# B&R Automation Studio project x20ost (part 7)

#### bnrdevts.c
```c
/********************************************************************
 * COPYRIGHT -- Kontora
 ********************************************************************
 * Program: bnrmain
 * File: bnrlsens.c
 * Author: Abramenya
 * Created: January 19, 2009
 *******************************************************************/

#include "bnrdevts.h"
#include "bnrmain.h"
#ifdef _DEFAULT_INCLUDES
 #include <AsDefault.h>
#endif
_GLOBAL BYTE nFSignal;
void CDevTS_Init(This,CPin *pPN,BOOL *pTlValue,BYTE byID,BYTE byIID,BYTE byState,BYTE byPriority,BYTE byCRemPulce,BYTE byCSetPulce,BYTE byAlarmMode)
{
    DECLARE_SINGLE_OPEN(CDevTS)
	//memcpy(pTU,&pT->pP,sizeof(STUMPARAM));
	pT->m_pPN          = pPN;
	pT->pP.byID        = byID;
	pT->pP.byAmParam   = byIID;
    pT->pP.byState     = byState;
    pT->pP.byPriority  = byPriority;
    pT->pP.byCRemPulce = byCRemPulce;
	pT->pP.byCSetPulce = byCSetPulce;
	pT->pP.byAlarmMode = byAlarmMode;

	pT->m_blTmSetState = FALSE;
	pT->m_blTmRemState = FALSE;
	pT->m_byType       = REG_SOFTS_ADDR;
	pT->m_blFSignal    = FALSE;

	pT->m_pTIN         = pTlValue;
	pT->m_byID         = pT->pP.byID;
    pT->m_byPinID      = pT->pP.byAmParam;
	pT->m_byOldEvent   = 0xff;
}
void CDevTS_SetTS(This,BYTE byBox,BYTE byFor,BYTE byEv)
{
    DECLARE_SINGLE_OPEN(CDevTS)
	pT->m_byBox  = byBox;
	pT->m_byFor  = byFor;
	pT->m_byEv   = byEv;
}
void CDevTS_PreProc(This)
{
    DECLARE_SINGLE_OPEN(CDevTS)
}
_GLOBAL INT nTSCH;
void CDevTS_Processing(This)
{
	DECLARE_SINGLE_OPEN(CDevTS)
	BYTE byState;
	if (pT->m_byID==40)	nTSCH++;
	if (pT->pP.byState==EN_OPEN)
	{
	 byState = pT->CheckTS(pT);
	 if(byState==PIN_STATE_ONN)
	 {
		 pT->m_blTmSetState = TRUE;pT->m_blTmRemState = FALSE;pT->m_bySetPulce = pT->pP.byCSetPulce;}
	 if(byState==PIN_STATE_OFF)
	 {
		 pT->m_blTmRemState = TRUE;pT->m_blTmSetState = FALSE;pT->m_byRemPulce = pT->pP.byCRemPulce;}
	 pT->pP.sDT.byParam = *pT->m_pTIN;
	}
}
void CDevTS_PostProc(This)
{
	DECLARE_SINGLE_OPEN(CDevTS)
	BOOL res = FALSE;
	//Set Timer
	if (pT->pP.byState==EN_OPEN)
	{
	if(pT->m_blTmSetState==TRUE)
	{
	 if (--pT->m_bySetPulce==0)
	 {
	  if((pT->pP.byPriority==PRI_HI)&&((pT->pP.byAlarmMode==EN_AL_TO_AL)||(pT->pP.byAlarmMode==EN_LO_TO_HI))) res = TRUE;
	  pT->SaveChange(pT,EV_0T1_CH,1,res);
	  pT->m_blTmSetState = FALSE;
	 }
	}
    //Rem Timer
	if(pT->m_blTmRemState==TRUE)
	{
	 if (--pT->m_byRemPulce==0)
	 {
	  if((pT->pP.byPriority==PRI_HI)&&((pT->pP.byAlarmMode==EN_AL_TO_AL)||(pT->pP.byAlarmMode==EN_HI_TO_LO))) res = TRUE;
	  if( pT->m_blFSignal)pT->SaveChange(pT,EV_1T0_CH,0,res);
	  pT->m_blTmRemState = FALSE;
	  pT->m_blFSignal = TRUE;
	 }
	}
	}
}
/*
typedef struct _tagKpEvent
{
WORD wLen;
BYTE byType;
BYTE byAddr;
BYTE byCause;
WORD wValue;
STIME sTime;
}SKPEVENT;
*/
BOOL CDevTS_SaveChange(This,BYTE byEvent,WORD wValue,BOOL blAlarm)
{
    DECLARE_SINGLE_OPEN(CDevTS)
	SKPEVENT sEV;
    if((byEvent!=pT->m_byOldEvent)||(byEvent==EV_CHG_PR))
	{
   	 pT->m_byOldEvent = byEvent;
	 sEV.wLen         = sizeof(SKPEVENT);
     sEV.byType       = pT->m_byType;
	 sEV.byCause      = byEvent;
	 sEV.wValue       = wValue;
	 sEV.byAddr       = pT->m_byPinID;
     if(blAlarm)
	 pT->SendEvent(pT,&sEV);
	}
	return TRUE;
}
void CDevTS_SendEvent(This,SKPEVENT *pEV)
{
    DECLARE_SINGLE_OPEN(CDevTS)
	SHORTMESSAGE m_sMsg	;
	m_sMsg.m_swLen        = 9 + sizeof(SKPEVENT);
	m_sMsg.m_sbyFrom      = pT->m_byFor;
	m_sMsg.m_sbyFor       = pT->m_byFor;
	m_sMsg.m_sbyIntType   = 0;
	m_sMsg.m_sbyServerID  = 0;
	m_sMsg.m_sbyType      = pT->m_byEv;
	m_sMsg.m_sbyDirection = 0;
	m_sMsg.m_sbySensor    = pT->m_byID;
	memcpy(&m_sMsg.m_sbyInfo[0],pEV,sizeof(SKPEVENT));
	FPUT(pT->m_byBox,(BYTE*)&m_sMsg);
}
BYTE CDevTS_CheckTS(This)
{
    DECLARE_SINGLE_OPEN(CDevTS)
	return pT->m_pPN->GetState(pT->m_pPN);
}
void CDevTS_Run(This)
{
    DECLARE_SINGLE_OPEN(CDevTS)
	pT->PreProc(pT);
	pT->Processing(pT);
	pT->PostProc(pT);
}
void CDevTS_CDevTS(This)
{
    DECLARE_SINGLE_OPEN(CDevTS)
	DECLARE_REGISTRATION(CDevTS,SaveChange)
	DECLARE_REGISTRATION(CDevTS,SendEvent)
	DECLARE_REGISTRATION(CDevTS,CheckTS)
	DECLARE_REGISTRATION(CDevTS,SetTS)
	DECLARE_REGISTRATION(CDevTS,Init)
	DECLARE_REGISTRATION(CDevTS,Run)
	DECLARE_REGISTRATION(CDevTS,PreProc)
	DECLARE_REGISTRATION(CDevTS,Processing)
	DECLARE_REGISTRATION(CDevTS,PostProc)
}
void CDevTS_DCDevTS(This)
{
	DECLARE_SINGLE_OPEN(CDevTS)
}
DECLARE_SINGLE_CREATE(CDevTS)
```

#### bnrdevts.h
```c
/********************************************************************
 * COPYRIGHT -- Kontora
 ********************************************************************
 * Program: bnrmain
 * File: bnraninput.h
 * Author: Abramenya
 * Created: January 19, 2009
 *******************************************************************/

#ifndef __DEVTS_H__
#define __DEVTS_H__
#include "typedefs.h"
#include "bnrtelesensor.h"
#include "bnrpin.h"
#define DEF_SET_PULSE 5
#define DEF_REM_PULSE 5
/*
STSMPARAMS nTS = {16,TS,{
{29  ,0 ,TS ,7 ,8 , 0, EN_OPEN, PRI_HI, 5, 5, EN_AL_TO_AL, 1},
typedef struct _tagTSMParam
{
BYTE byID;
BYTE byAmParam;
BYTE byType;
BYTE bySlot;
BYTE byPin;
BYTE byAlmState;
BYTE byState;
BYTE byPriority;
BYTE byCRemPulce;
BYTE byCSetPulce;
BYTE byAlarmMode;
STSMDATA sDT;
}STSMPARAM;
*/
Class CDevTS
{
	 void (*CCDevTS)(This);
	 void (*DCDevTS)(This);
Public
     BYTE (*CheckTS)(This);
     void (*Init)(This,CPin *pPN,BOOL *pblValue,BYTE byID,BYTE byIID,BYTE byState,BYTE byPriority,BYTE byCRemPulce,BYTE byCSetPulce,BYTE byAlarmMode);
	 void (*SetTS)(This,BYTE byBox,BYTE byFor,BYTE byEv);
     void (*PreProc)(This);
     void (*Processing)(This);
	 void (*PostProc)(This);
	 void (*SendEvent)(This,SKPEVENT *pEV);
	 BOOL (*SaveChange)(This,BYTE byEvent,WORD wValue,BOOL blAlarm);
	 void (*Run)(This);
Public
     STSMPARAM pP;
     BYTE m_byBox;
     BYTE m_byFor;
     BYTE m_byEv;
     BYTE m_byID;
	 BYTE m_byPinID;
	 BYTE m_byOldEvent;

	 BOOL *m_pTIN;
	 BOOL m_blFSignal;
     BOOL m_blTmSetState;
	 BOOL m_blTmRemState;
     BYTE m_bySetPulce;
	 BYTE m_byRemPulce;
	 BYTE m_byType;
	 CPin *m_pPN;
	 DECLARE_IMPLEMENT
}
DECLARE_DEFINITION(CDevTS)
#endif
```

#### bnrdevtu.c
```c
/********************************************************************
 * COPYRIGHT -- Kontora
 ********************************************************************
 * Program: bnrmain
 * File: bnrlsens.c
 * Author: Abramenya
 * Created: January 19, 2009
 *******************************************************************/

#include "bnrdevtu.h"
#ifdef _DEFAULT_INCLUDES
#include <AsDefault.h>
#endif
/*
BYTE byID;
    BYTE byAmParam;
	STUMPARAMS nTU = {10,TU,{
	{45  ,0 ,TU ,10, 2 , 0, EN_OPEN, EN_DIRECT, 5, 1},
	typedef struct _tagTUMParam
	{
	BYTE byID;
	BYTE byAmParam;
	BYTE byType;
	BYTE bySlot;
	BYTE byPin;
	BYTE byAlmState;
	BYTE byState;
	BYTE byPulceType;
    WORD byCSetPulce;
	STUMDATA sDT;
}STUMPARAM;
*/
void CDevTU_Init(This,BOOL *pblValue,BYTE byID,BYTE byIID,BYTE byState,BYTE byPulceType,DWORD byCSetPulce)
{
    DECLARE_SINGLE_OPEN(CDevTU)
	//memcpy(pTU,&pT->pP,sizeof(STUMPARAM));
	pT->pP.byID        = byID;
	pT->pP.byAmParam   = byIID;
    pT->pP.byState     = byState;
    pT->pP.byPulceType = byPulceType;
    pT->pP.byCSetPulce = byCSetPulce;
	pT->m_dwJob        = byPulceType;

	pT->m_pbOT       = pblValue;
	pT->m_byType     = REG_SOFTU_ADDR;
	pT->m_byStPulce  = FALSE;
	pT->m_byID       = pT->pP.byID;
    pT->m_byPinID    = pT->pP.byAmParam;
	pT->m_byOldEvent = 0xff;
	//pT->InvPin(pT);
	//if (pT->pP.byPulceType==EN_DIRECT) *pT->m_pbOT = FALSE; else
	//if (pT->pP.byPulceType==EN_INVERT) *pT->m_pbOT = TRUE;
}
void CDevTU_SetTU(This,BYTE byBox,BYTE byFor,BYTE byEv)
{
    DECLARE_SINGLE_OPEN(CDevTU)
	pT->m_byBox  = byBox;
	pT->m_byFor  = byFor;
	pT->m_byEv   = byEv;
}
void CDevTU_PreProc(This)
{
    DECLARE_SINGLE_OPEN(CDevTU)
}
_GLOBAL INT nTCCH;
void CDevTU_Processing(This)
{
	DECLARE_SINGLE_OPEN(CDevTU)
	if (pT->m_byID==5)	nTCCH++;
	if(pT->pP.byState==EN_OPEN)
	{
	 if(pT->m_byStPulce==TRUE)
	 {
	 if (--pT->m_bySetPulce==0)
	 {
	   if(*pT->m_pbOT==FALSE)
	   {
	   *pT->m_pbOT = TRUE;
	   pT->SaveChange(pT,EV_0T1_ST,1,FALSE);
	   }else
	   if(*pT->m_pbOT==TRUE )
	   {
	   *pT->m_pbOT = FALSE;
	   pT->SaveChange(pT,EV_1T0_ST,0,FALSE);
	   }
       #ifdef DEB_CDevTU
	   Info("\n(%b)CTLCT::>SetPulce::STOP.",&pT->m_byID);
       #endif
	   pT->m_byStPulce  = FALSE;
	 }
	 }
	 pT->pP.sDT.byParam = *pT->m_pbOT;
	}
}
void CDevTU_PostProc(This)
{
	DECLARE_SINGLE_OPEN(CDevTU)
}
void CDevTU_Stop(This)
{
    DECLARE_SINGLE_OPEN(CDevTU)
    if(pT->pP.byState==EN_OPEN)
	{
	if(pT->m_byStPulce==TRUE)
	{
	  pT->m_bySetPulce = pT->pP.byCSetPulce;
	  pT->m_dwJob      = pT->pP.byCSetPulce;
	  pT->m_bySetPulce = 0;
	  pT->m_byStPulce  = FALSE;
	  if(*pT->m_pbOT==FALSE)
	  {
	   *pT->m_pbOT = TRUE;
	   pT->SaveChange(pT,EV_0T1_ST,1,FALSE);
	  }else
	  if(*pT->m_pbOT==TRUE )
	  {
	   *pT->m_pbOT = FALSE;
	   pT->SaveChange(pT,EV_1T0_ST,0,FALSE);
	  }
	 #ifdef DEB_CDevTU
	 Info("\n(%b)CTLCT::>StopPulce",&pT->m_byID);
     #endif
	}
	}
}
void CDevTU_PreparePulce(This)
{
    DECLARE_SINGLE_OPEN(CDevTU)
	if(pT->pP.byState==EN_OPEN)
	{
	 //pT->m_bySetPulce = pT->pP.byCSetPulce;
	 pT->m_byStPulce  = TRUE;
	 if (pT->pP.byPulceType==EN_DIRECT)
	 {
	  *pT->m_pbOT = TRUE;
	  pT->SaveChange(pT,EV_0T1_ST,1,FALSE);
	 }
	 if (pT->pP.byPulceType==EN_INVERT)
	 {
	  *pT->m_pbOT = FALSE;
	  pT->SaveChange(pT,EV_1T0_ST,0,FALSE);
	 }
	 #ifdef DEB_CDevTU
	 Info("\n(%b)CTLCT::>SetPulce::START.",&pT->m_byID);
     #endif
	}
}
void CDevTU_SetPulce(This)
{
    DECLARE_SINGLE_OPEN(CDevTU)
    pT->m_bySetPulce = pT->pP.byCSetPulce;
	pT->m_dwJob      = pT->pP.byCSetPulce;
	pT->PreparePulce(pT);
}
void CDevTU_SetPulceEx(This,DWORD dwPulce)
{
    DECLARE_SINGLE_OPEN(CDevTU)
    pT->m_bySetPulce = dwPulce;
	pT->m_dwJob      = dwPulce;
	pT->PreparePulce(pT);
}
void CDevTU_SetPin(This)
{
    DECLARE_SINGLE_OPEN(CDevTU)
	if(pT->pP.byState==EN_OPEN)
	{
	 //pT->m_bySetPulce = pT->pP.byCSetPulce;
	 //pT->m_byStPulce  = TRUE;
	 if (pT->pP.byPulceType==EN_DIRECT)
	 {
	  *pT->m_pbOT = TRUE;
	  pT->SaveChange(pT,EV_0T1_ST,1,FALSE);
	 }
	 if (pT->pP.byPulceType==EN_INVERT)
	 {
	  *pT->m_pbOT = FALSE;
	  pT->SaveChange(pT,EV_1T0_ST,0,FALSE);
	 }
	 pT->pP.sDT.byParam = *pT->m_pbOT;
	 #ifdef DEB_CDevTU
	 Info("\n(%b)CTLCT::>SetPulce::START.",&pT->m_byID);
     #endif
	}
}
void CDevTU_InvPin(This)
{
    DECLARE_SINGLE_OPEN(CDevTU)
	if(pT->pP.byState==EN_OPEN)
	{
	 //pT->m_bySetPulce = pT->pP.byCSetPulce;
	 //pT->m_byStPulce  = TRUE;
	 if (pT->pP.byPulceType==EN_DIRECT)
	 {
	  *pT->m_pbOT = FALSE;
	  pT->SaveChange(pT,EV_1T0_ST,0,FALSE);
	 }
	 if (pT->pP.byPulceType==EN_INVERT)
	 {
	  *pT->m_pbOT = TRUE;
	  pT->SaveChange(pT,EV_0T1_ST,1,FALSE);
	 }
	 pT->pP.sDT.byParam = *pT->m_pbOT;
	 #ifdef DEB_CDevTU
	 Info("\n(%b)CTLCT::>InvPulce::START.",&pT->m_byID);
     #endif
	}
}
/*
typedef struct _tagKpEvent
{
WORD wLen;
BYTE byType;
BYTE byAddr;
BYTE byCause;
WORD wValue;
STIME sTime;
}SKPEVENT;
*/
BOOL CDevTU_SaveChange(This,BYTE byEvent,WORD wValue,BOOL blAlarm)
{
    DECLARE_SINGLE_OPEN(CDevTU)
	SKPEVENT sEV;
    if((byEvent!=pT->m_byOldEvent)||(byEvent==EV_CHG_PR))
	{
   	 pT->m_byOldEvent = byEvent;
	 sEV.wLen         = sizeof(SKPEVENT);
     sEV.byType       = pT->m_byType;
	 sEV.byCause      = byEvent;
	 sEV.wValue       = wValue;
	 sEV.byAddr       = pT->m_byPinID;
     if(!blAlarm)
	 pT->SendEvent(pT,&sEV);
	}
	return TRUE;
}
void CDevTU_SendEvent(This,SKPEVENT *pEV)
{
    DECLARE_SINGLE_OPEN(CDevTU)
	SHORTMESSAGE m_sMsg	;
	m_sMsg.m_swLen        = 9 + sizeof(SKPEVENT);
	m_sMsg.m_sbyFrom      = pT->m_byFor;
	m_sMsg.m_sbyFor       = pT->m_byFor;
	m_sMsg.m_sbyIntType   = 0;
	m_sMsg.m_sbyServerID  = 0;
	m_sMsg.m_sbyType      = pT->m_byEv;
	m_sMsg.m_sbyDirection = 0;
	m_sMsg.m_sbySensor    = pT->m_byID;
	memcpy(&m_sMsg.m_sbyInfo[0],pEV,sizeof(SKPEVENT));
	FPUT(pT->m_byBox,(BYTE*)&m_sMsg);
}
DWORD CDevTU_Run(This)
{
    DECLARE_SINGLE_OPEN(CDevTU)
	DWORD dwRes=0;
	pT->PreProc(pT);
	pT->Processing(pT);
	pT->PostProc(pT);
	if ((pT->m_dwJob>=pT->m_bySetPulce)&&(pT->m_bySetPulce!=0)) dwRes = pT->m_dwJob-pT->m_bySetPulce;
	return dwRes;
}
void CDevTU_CDevTU(This)
{
    DECLARE_SINGLE_OPEN(CDevTU)
	DECLARE_REGISTRATION(CDevTU,SetPulce)
	DECLARE_REGISTRATION(CDevTU,Stop)
	DECLARE_REGISTRATION(CDevTU,SetPulceEx)
	DECLARE_REGISTRATION(CDevTU,PreparePulce)
	DECLARE_REGISTRATION(CDevTU,SaveChange)
	DECLARE_REGISTRATION(CDevTU,SendEvent)
	DECLARE_REGISTRATION(CDevTU,SetTU)
	DECLARE_REGISTRATION(CDevTU,SetPin)
	DECLARE_REGISTRATION(CDevTU,InvPin)
	DECLARE_REGISTRATION(CDevTU,Init)
	DECLARE_REGISTRATION(CDevTU,Run)
	DECLARE_REGISTRATION(CDevTU,PreProc)
	DECLARE_REGISTRATION(CDevTU,Processing)
	DECLARE_REGISTRATION(CDevTU,PostProc)
}
void CDevTU_DCDevTU(This)
{
	DECLARE_SINGLE_OPEN(CDevTU)
}
DECLARE_SINGLE_CREATE(CDevTU)
```

#### bnrdvs.h
```c
/********************************************************************
 * COPYRIGHT -- Kontora
 ********************************************************************
 * Program: bnrmain
 * File: bnraninput.h
 * Author: Abramenya
 * Created: January 19, 2009
 *******************************************************************/

#ifndef __DVS_H__
#define __DVS_H__
#include "typedefs.h"
#include "bnrdevice.h"
#include "bnrpin.h"

Class CDvs
{
	 void (*CCDvs)(This);
	 void (*DCDvs)(This);
Public
     BYTE (*CheckTS)(This);
	 Virtual BOOL (*EventHandler)(This,SMESSAGE *pMsg);
	 Virtual void (*InitTCHN)(This,PVOID psTable);
     Virtual void (*PreProc)(This);
	 Virtual void (*Processing)(This);
     Virtual void (*PostProc)(This);
	 Virtual void (*SetInPinEvent)(This);
	 Virtual void (*SaveAlarmPin)(This);
	 Virtual void (*SendObsrveMsg)(This);
	 Virtual PVOID (*GetData)(This,BYTE *pData,WORD *nLen);
Public
     STVSPARAM *pP;
	 DECLARE_IMPLEMENT_BASE(CDevice)
}
DECLARE_DEFINITION(CDvs)
#endif
```

#### bnrdvs.c
```c
/********************************************************************
 * COPYRIGHT -- Kontora
 ********************************************************************
 * Program: bnrmain
 * File: bnrlsens.c
 * Author: Abramenya
 * Created: January 19, 2009
 *******************************************************************/

#include "bnrdvs.h"
#include "bnrmain.h"
#ifdef _DEFAULT_INCLUDES
 #include <AsDefault.h>
#endif
_GLOBAL BYTE nFSignal;
SINT *chDV[] =
{
	"010.145000",
};
void CDvs_InitTCHN(This,PVOID psTable)
{
    DECLARE_MULTI_OPEN(CDvs,CDevice)
	pT->pP = (STVSPARAM*)psTable;
	pB->m_nSize = 11;
	strcpy(pT->pP->sDT.byData,chDV[0]);
    #ifdef DEB_CDvs
	//Info("\n(%b)CTLSG::>Create TeleSignal.",&pB->m_byID);
    #endif
}
void CDvs_PreProc(This)
{
    DECLARE_MULTI_OPEN(CDvs,CDevice)

}
_GLOBAL INT nTSCH;
void CDvs_Processing(This)
{
	DECLARE_MULTI_OPEN(CDvs,CDevice)
}
void CDvs_PostProc(This)
{
	DECLARE_MULTI_OPEN(CDvs,CDevice)
}
BYTE CDvs_CheckTS(This)
{
    DECLARE_MULTI_OPEN(CDvs,CDevice)
	//return pB->m_pPN->GetState(pB->m_pPN);
	return 0;
}
BOOL CDvs_EventHandler(This,SMESSAGE *pMsg)
{
    DECLARE_MULTI_OPEN(CDvs,CDevice)
    BYTE byID = pMsg->m_sbySensor;
	BYTE byParamType = pMsg->m_sbyInfo[3];
    #ifdef DEB_CDvs
	Info("\n(%b)CTLSG::>INPT::%M",&pB->m_byID,pMsg);
    #endif
	switch(pMsg->m_sbyFor)
	{
	  case DIR_101TOKP:
		   switch(pMsg->m_sbyType)
		   {
		    case PL_DATA_IND:
				 //Info("\n(%b)CTLSG::>DL_DATA_IND::>%M",&pB->m_byID,pMsg);
				 switch(byParamType)
				 {
				   case EN_SET_PERIOD:
					    //pT->m_byCSetPulce = pMsg->m_sbyInfo[3];
					    //pT->m_bySetPulce  = pT->m_byCSetPulce;
				   break;
				   case EN_REM_PERIOD:
					    //pT->m_byRemPulce  = pMsg->m_sbyInfo[3];
						//pT->m_byCRemPulce = pT->m_byRemPulce;
				   break;
				   case EN_PIN_ALMODE:
                        //pT->m_byAlarmMode = pMsg->m_sbyInfo[3];
				   break;
				   default:
				   break;
				 }
		    break;
			default:
            break;
		   }
      break;
	  case DIR_101MD:
	  break;
	  default:
	  break;
	}
	return TRUE;
}
void CDvs_SetInPinEvent(This)
{
    DECLARE_MULTI_OPEN(CDvs,CDevice)
}
void CDvs_SaveAlarmPin(This)
{
	DECLARE_MULTI_OPEN(CDvs,CDevice)
}
void CDvs_SendObsrveMsg(This)
{
    DECLARE_MULTI_OPEN(CDvs,CDevice)
}
/*
typedef struct _tagTVSData
{
BYTE byData[11];
}STVSDATA;
*/
PVOID CDvs_GetData(This,BYTE *pData,WORD *nLen)
{
    DECLARE_MULTI_OPEN(CDvs,CDevice)
	memcpy(pData,&pT->pP->sDT.byData[0],11);
	*nLen += pB->m_nSize;if (*nLen>350) *nLen=0;
	return pData;
}
void CDvs_CDvs(This)
{
    DECLARE_MULTI_OPEN(CDvs,CDevice)
	DECLARE_REGISTRATION(CDvs,CheckTS)
	DECLARE_VIRTUAL_FUNC(CDvs,EventHandler)
	DECLARE_VIRTUAL_FUNC(CDvs,InitTCHN)
	DECLARE_VIRTUAL_FUNC(CDvs,PreProc)
	DECLARE_VIRTUAL_FUNC(CDvs,Processing)
	DECLARE_VIRTUAL_FUNC(CDvs,PostProc)
	DECLARE_VIRTUAL_FUNC(CDvs,SetInPinEvent)
	DECLARE_VIRTUAL_FUNC(CDvs,SaveAlarmPin)
	DECLARE_VIRTUAL_FUNC(CDvs,SendObsrveMsg)
	DECLARE_VIRTUAL_FUNC(CDvs,GetData)
}
void CDvs_DCDvs(This)
{
	DECLARE_MULTI_OPEN(CDvs,CDevice)
}
DECLARE_MULTI_CREATE(CDvs,CDevice)
```

#### bnrfreq.h
```c
/********************************************************************
 * COPYRIGHT -- Kontora
 ********************************************************************
 * Program: bnrmain
 * File: bnraninput.h
 * Author: Abramenya
 * Created: January 19, 2009
 *******************************************************************/

#ifndef __FREQ_H__
#define __FREQ_H__
#include "typedefs.h"
#include "bnrdevice.h"
#include "bnrpin.h"
#include "bnrdevtu.h"
#include "bnrdevts.h"
Class CFreq
{
	 void (*CCFreq)(This);
	 void (*DCFreq)(This);
Public
     void (*StartFC)(This);
     void (*StopFC)(This);
	 Virtual BOOL (*EventHandler)(This,SMESSAGE *pMsg);
	 Virtual void (*InitTCHN)(This,PVOID psTable);
     Virtual void (*PreProc)(This);
	 Virtual void (*Processing)(This);
     Virtual void (*PostProc)(This);
	 Virtual PVOID (*GetData)(This,BYTE *pData,WORD *nLen);
Public
     STFPARAM *pP;
     CDevTU *pTU0;
     CDevTU *pTU1;
	 CDevTS *pTS0;
	 CDevTS *pTS1;
     WORD *m_pwVL0;
	 DECLARE_IMPLEMENT_BASE(CDevice)
}
DECLARE_DEFINITION(CFreq)
#endif
```

#### bnrfreq.c
```c
/********************************************************************
 * COPYRIGHT -- Kontora
 ********************************************************************
 * Program: bnrmain
 * File: bnrlsens.c
 * Author: Abramenya
 * Created: January 19, 2009
 *******************************************************************/

#include "bnrfreq.h"
#include "bnrmain.h"
#ifdef _DEFAULT_INCLUDES
 #include <AsDefault.h>
#endif
_GLOBAL BYTE nFSignal;
/*
typedef struct _tagTFParam
{
BYTE byID;
BYTE byAmParam;
BYTE byType;
BYTE bySlot; //Для задания
BYTE byPin;  //Для задания

  BYTE bySlot1; //Запуск
  BYTE byPin1;  //Запуск

	BYTE bySlot2; //Останов
	BYTE byPin2;  //Останов

	  BYTE bySlot3; //Авария1
	  BYTE byPin3;  //Авария1

		BYTE bySlot4; //Авария2
		BYTE byPin4;  //Авария2
		STFDATA sDT;
}STFPARAM;
*/
void CFreq_InitTCHN(This,PVOID psTable)
{
    DECLARE_MULTI_OPEN(CFreq,CDevice)
	CSlot *pSL;
	CPin *m_pPN0;
	BOOL *m_pbVL0;
	BOOL *m_pbVL1;
	BOOL *m_pbAVL0;
	BOOL *m_pbAVL1;
	CComputer *pCM = pB->m_pComputer;
    pT->pP = (STFPARAM*)psTable;
	pB->m_nSize = 3*sizeof(WORD);
    //Задание
	pSL          = pCM->GetSlot(pCM,pT->pP->bySlot);
	m_pPN0       = pSL->GetPin(pSL->pChld,pT->pP->byPin);
    pT->m_pwVL0 = (WORD*)m_pPN0->GetAddrPin(m_pPN0->pChld);

    //Выход запуска
	pSL          = pCM->GetSlot(pCM,pT->pP->bySlot1);
	m_pPN0       = pSL->GetPin(pSL->pChld,pT->pP->byPin1);
    m_pbVL0 = (BOOL*)m_pPN0->GetAddrPin(m_pPN0->pChld);
	New(sizeof(CDevTU),pT->pTU0);
	InitObject(CDevTU,pT->pTU0);
    pT->pTU0->Init(pT->pTU0,m_pbVL0,pT->pP->byID,0,EN_OPEN,EN_DIRECT,10);
	pT->pTU0->SetTU(pT->pTU0,DEV_MSMDL_BOX_ID,DIR_MSTOMS,EV_CHNG_PIN_REQ);

	//Выход останова
	pSL          = pCM->GetSlot(pCM,pT->pP->bySlot2);
	m_pPN0       = pSL->GetPin(pSL->pChld,pT->pP->byPin2);
    m_pbVL1 = (BOOL*)m_pPN0->GetAddrPin(m_pPN0->pChld);

	New(sizeof(CDevTU),pT->pTU1);
	InitObject(CDevTU,pT->pTU1);
    pT->pTU1->Init(pT->pTU1,m_pbVL1,pT->pP->byID,1,EN_OPEN,EN_DIRECT,10);
	pT->pTU1->SetTU(pT->pTU1,DEV_MSMDL_BOX_ID,DIR_MSTOMS,EV_CHNG_PIN_REQ);

	//Вход активности
	pSL          = pCM->GetSlot(pCM,pT->pP->bySlot3);
	m_pPN0       = pSL->GetPin(pSL->pChld,pT->pP->byPin3);
    m_pbAVL0 = (BOOL*)m_pPN0->GetAddrPin(m_pPN0->pChld);

	New(sizeof(CDevTS),pT->pTS0);
	InitObject(CDevTS,pT->pTS0);
    pT->pTS0->Init(pT->pTS0,m_pPN0, m_pbAVL0,pT->pP->byID,0,EN_OPEN,PRI_HI,10,10,EN_AL_TO_AL);
	pT->pTS0->SetTS(pT->pTS0,DEV_MSMDL_BOX_ID,DIR_MSTOMS,EV_CHNG_PIN_REQ);

	//Вход Аварии
	pSL          = pCM->GetSlot(pCM,pT->pP->bySlot4);
	m_pPN0       = pSL->GetPin(pSL->pChld,pT->pP->byPin4);
    m_pbAVL1 = (BOOL*)m_pPN0->GetAddrPin(m_pPN0->pChld);

	New(sizeof(CDevTS),pT->pTS1);
	InitObject(CDevTS,pT->pTS1);
    pT->pTS1->Init(pT->pTS1,m_pPN0, m_pbAVL1,pT->pP->byID,1,EN_OPEN,PRI_HI,10,10,EN_AL_TO_AL);
	pT->pTS1->SetTS(pT->pTS1,DEV_MSMDL_BOX_ID,DIR_MSTOMS,EV_CHNG_PIN_REQ);

    #ifdef DEB_CFreq
	//Info("\n(%b)CTLSG::>Create TeleSignal.",&pB->m_byID);
    #endif
}
void CFreq_PreProc(This)
{
    DECLARE_MULTI_OPEN(CFreq,CDevice)
	pT->pTU0->Run(pT->pTU0);
	pT->pTU1->Run(pT->pTU1);
	pT->pTS0->Run(pT->pTS0);
	pT->pTS1->Run(pT->pTS1);
}
_GLOBAL INT nTSCH;
void CFreq_Processing(This)
{
	DECLARE_MULTI_OPEN(CFreq,CDevice)
}
void CFreq_PostProc(This)
{
	DECLARE_MULTI_OPEN(CFreq,CDevice)
}
/*
typedef struct _tagTFData
{
BYTE byStartST;
BYTE byStopST;
BYTE byAlST0;
BYTE byAlST1;
WORD wTask;
WORD wParam;
}STFDATA;
typedef struct _tagKpEvent
{
WORD wLen;
BYTE byType;
BYTE byAddr;
BYTE byCause;
WORD wValue;
STIME sTime;
}SKPEVENT;
*/
BOOL CFreq_EventHandler(This,SMESSAGE *pMsg)
{
    DECLARE_MULTI_OPEN(CFreq,CDevice)
	SKPEVENT pEV;
    #ifdef DEB_CFreq
	Info("\n(%b)CTLSG::>INPT::%M",&pB->m_nCD.wDeviceID,pMsg);
    #endif
	switch(pMsg->m_sbyFor)
	{
	  case DIR_MSTODV:
		   switch(pMsg->m_sbyType)
		   {
		    case PL_DATA_IND:
				 switch(pB->m_nCD.byParam0)
				 {
				   case CTR_TR:
                        //#ifdef DEB_CFreq
	                    //Info("\n(%b)CTLSG::>CTR_TR::%d",&pB->m_nCD.wDeviceID,&pB->m_nCD.fParam0);
                        //#endif
						pT->pP->sDT.wTask = (WORD)pB->m_nCD.fParam0;
						*pT->m_pwVL0      = (WORD)pB->m_nCD.fParam0;
				   break;
				   case CTR_TU:
					   switch (pB->m_nCD.byParam1)
					   {
					      case 0:
					         if (pB->m_nCD.wParam0==1) pT->StartFC(pT);else
					         if (pB->m_nCD.wParam0==0) pT->StopFC(pT);
						  break;
						  case 1:
							  if (pB->m_nCD.wParam0==0)
							  {
							   pT->pP->sDT.wSt0 &= ~(0x02);
							   pT->pTU0->InvPin(pT->pTU0);
                               pT->pTU1->SetPin(pT->pTU1);
							  }
							  else
							  if (pB->m_nCD.wParam0==1) pT->pP->sDT.wSt0 |=  (0x02);
						  break;
						  default:
						  break;
					   }
                        //#ifdef DEB_CFreq
	                    //Info("\n(%b)CTLSG::>CTR_TR::%d",&pB->m_nCD.wDeviceID,&pB->m_nCD.fParam0);
                        //#endif
				   break;
				   default:
				   break;
				 }
		    break;
			case EV_CHNG_PIN_REQ:
 				 memcpy(&pEV,&pMsg->m_sbyInfo[0],sizeof(SKPEVENT));
				 switch (pEV.byType)
				 {
				    case REG_SOFTU_ADDR:
						if ((pEV.byCause==EV_0T1_ST)&&(pEV.byAddr==0))
							pT->pP->sDT.wSt0 |=  (0x01);
						if ((pEV.byCause==EV_1T0_ST)&&(pEV.byAddr==0))
							pT->pP->sDT.wSt0 &= ~(0x01);
					break;
					case REG_SOFTS_ADDR:
						//Активность с релейного выхода
						if ((pEV.byCause==EV_0T1_CH)&&(pEV.byAddr==0))
							pT->pP->sDT.wSt0 |=  (0x04);
						if ((pEV.byCause==EV_1T0_CH)&&(pEV.byAddr==0))
							pT->pP->sDT.wSt0 &= ~(0x04);
						//Авария
						if ((pEV.byCause==EV_0T1_CH)&&(pEV.byAddr==1))
							pT->pP->sDT.wSt0 |=  (0x08);
						if ((pEV.byCause==EV_1T0_CH)&&(pEV.byAddr==1))
							pT->pP->sDT.wSt0 &= ~(0x08);
					break;
				 }
			break;
			default:
            break;
		   }
      break;
	  case DIR_101MD:
	  break;
	  default:
	  break;
	}
	return TRUE;
}
void CFreq_StartFC(This)
{
    DECLARE_MULTI_OPEN(CFreq,CDevice)
	if(pT->pP->sDT.wSt0 & 0x02)
	{
	 pT->pTU0->SetPin(pT->pTU0);
	 pT->pTU1->InvPin(pT->pTU1);
	}
}
void CFreq_StopFC(This)
{
    DECLARE_MULTI_OPEN(CFreq,CDevice)
	if(pT->pP->sDT.wSt0 & 0x02)
	{
	 pT->pTU0->InvPin(pT->pTU0);
	 pT->pTU1->SetPin(pT->pTU1);
	}
}
/*
typedef struct _tagTFData
{
BYTE byStartST;
BYTE byStopST;
BYTE byAlST0;
BYTE byAlST1;
WORD wTask;
WORD wParam;
}STFDATA;
*/
PVOID CFreq_GetData(This,BYTE *pData,WORD *nLen)
{
    DECLARE_MULTI_OPEN(CFreq,CDevice)
	pB->GetWordParam(pB,(BYTE*)&pT->pP->sDT.wSt0,&pData[0]);
	pB->GetWordParam(pB,(BYTE*)&pT->pP->sDT.wTask,&pData[2]);
	pB->GetWordParam(pB,(BYTE*)&pT->pP->sDT.wParam,&pData[4]);
	*nLen += pB->m_nSize;if (*nLen>350) *nLen=0;
	return pData;
}
void CFreq_CFreq(This)
{
    DECLARE_MULTI_OPEN(CFreq,CDevice)
	DECLARE_REGISTRATION(CFreq,StartFC)
	DECLARE_REGISTRATION(CFreq,StopFC)
	DECLARE_VIRTUAL_FUNC(CFreq,EventHandler)
	DECLARE_VIRTUAL_FUNC(CFreq,InitTCHN)
	DECLARE_VIRTUAL_FUNC(CFreq,PreProc)
	DECLARE_VIRTUAL_FUNC(CFreq,Processing)
	DECLARE_VIRTUAL_FUNC(CFreq,PostProc)
	DECLARE_VIRTUAL_FUNC(CFreq,GetData)
}
void CFreq_DCFreq(This)
{
	DECLARE_MULTI_OPEN(CFreq,CDevice)
}
DECLARE_MULTI_CREATE(CFreq,CDevice)
```

#### bnrlevel.h
```c
/********************************************************************
 * COPYRIGHT -- Kontora
 ********************************************************************
 * Program: bnrmain
 * File: bnraninput.h
 * Author: Abramenya
 * Created: January 19, 2009
 *******************************************************************/

#ifndef __LEVEL_H__
#define __LEVEL_H__
#include "typedefs.h"
#include "bnrdevice.h"
#include "bnrpin.h"
#include "bnrdevtu.h"
#include "bnrdevts.h"
Class CLevel
{
	 void (*CCLevel)(This);
	 void (*DCLevel)(This);
Public
	 Virtual BOOL (*EventHandler)(This,SMESSAGE *pMsg);
	 Virtual void (*InitTCHN)(This,PVOID psTable);
     Virtual void (*PreProc)(This);
	 Virtual void (*Processing)(This);
     Virtual void (*PostProc)(This);
	 Virtual PVOID (*GetData)(This,BYTE *pData,WORD *nLen);
Public
     SLVPARAM *pP;
     CDevTS *pTS0;
     CDevTS *pTS1;
	 DECLARE_IMPLEMENT_BASE(CDevice)
}
DECLARE_DEFINITION(CLevel)
#endif
```

#### bnrlevel.c
```c
/********************************************************************
 * COPYRIGHT -- Kontora
 ********************************************************************
 * Program: bnrmain
 * File: bnrlsens.c
 * Author: Abramenya
 * Created: January 19, 2009
 *******************************************************************/

#include "bnrlevel.h"
#include "bnrmain.h"
#ifdef _DEFAULT_INCLUDES
 #include <AsDefault.h>
#endif
_GLOBAL BYTE nFSignal;
void CLevel_InitTCHN(This,PVOID psTable)
{
    DECLARE_MULTI_OPEN(CLevel,CDevice)
	CSlot *pSL;
	CPin *m_pPN0;
	BOOL *m_pbAVL0;
	CComputer *pCM = pB->m_pComputer;

    pT->pP = (SLVPARAM*)psTable;
	pB->m_nSize = 4*sizeof(WORD);

    //Вход нижнее положение
	pSL          = pCM->GetSlot(pCM,pT->pP->bySlot);
	m_pPN0       = pSL->GetPin(pSL->pChld,pT->pP->byPin);
    m_pbAVL0 = (BOOL*)m_pPN0->GetAddrPin(m_pPN0->pChld);
	New(sizeof(CDevTS),pT->pTS0);
	InitObject(CDevTS,pT->pTS0);
    pT->pTS0->Init(pT->pTS0,m_pPN0, m_pbAVL0,pT->pP->byID,0,EN_OPEN,PRI_HI,3,3,EN_AL_TO_AL);
	pT->pTS0->SetTS(pT->pTS0,DEV_MSMDL_BOX_ID,DIR_MSTOMS,EV_CHNG_PIN_REQ);

	//Вход верхнее положение
	pSL          = pCM->GetSlot(pCM,pT->pP->bySlot1);
	m_pPN0       = pSL->GetPin(pSL->pChld,pT->pP->byPin1);
    m_pbAVL0 = (BOOL*)m_pPN0->GetAddrPin(m_pPN0->pChld);
	New(sizeof(CDevTS),pT->pTS1);
	InitObject(CDevTS,pT->pTS1);
    pT->pTS1->Init(pT->pTS1,m_pPN0, m_pbAVL0,pT->pP->byID,1,EN_OPEN,PRI_HI,3,3,EN_AL_TO_AL);
	pT->pTS1->SetTS(pT->pTS1,DEV_MSMDL_BOX_ID,DIR_MSTOMS,EV_CHNG_PIN_REQ);
    #ifdef DEB_CLevel
	//Info("\n(%b)CTLSG::>Create TeleSignal.",&pB->m_byID);
    #endif
}
void CLevel_PreProc(This)
{
    DECLARE_MULTI_OPEN(CLevel,CDevice)
	pT->pTS0->Run(pT->pTS0);
	pT->pTS1->Run(pT->pTS1);
}
_GLOBAL INT nTSCH;
void CLevel_Processing(This)
{
	DECLARE_MULTI_OPEN(CLevel,CDevice)
}
void CLevel_PostProc(This)
{
	DECLARE_MULTI_OPEN(CLevel,CDevice)
	BOOL res = FALSE;
}
/*
typedef struct _tagLVData
{
WORD wSt0;
WORD wJob0;
WORD wJob1;
WORD wParam;
}SLVDATA;
*/
BOOL CLevel_EventHandler(This,SMESSAGE *pMsg)
{
    DECLARE_MULTI_OPEN(CLevel,CDevice)
	SKPEVENT pEV;
    #ifdef DEB_CLevel
	//Info("\n(%b)CTLSG::>INPT::%M",&pB->m_nCD.wDeviceID,pMsg);
    #endif
	switch(pMsg->m_sbyFor)
	{
	  case DIR_MSTODV:
		   switch(pMsg->m_sbyType)
		   {
		    case PL_DATA_IND:
				 switch(pB->m_nCD.byParam0)
				 {
                   case CTR_TR:
					    switch (pB->m_nCD.byParam1)
					    {
						  case 0:
							  if ((WORD)pB->m_nCD.fParam0>pT->pP->sDT.wJob1)
							  pT->pP->sDT.wJob0 = (WORD)(pB->m_nCD.fParam0);
						  break;
						  case 1:
							  if ((WORD)pB->m_nCD.fParam0<pT->pP->sDT.wJob0)
							  pT->pP->sDT.wJob1 = (WORD)(pB->m_nCD.fParam0);
						  break;
						  default:
						  break;
					    }
				   break;
				   case CTR_TU:
				   break;
				   default:
				   break;
				 }
		    break;
			case EV_CHNG_PIN_REQ:
 				 memcpy(&pEV,&pMsg->m_sbyInfo[0],sizeof(SKPEVENT));
				 switch (pEV.byType)
				 {
				    case REG_SOFTU_ADDR:
						//if ((pEV.byCause==EV_0T1_ST)&&(pEV.byAddr==0))
						//	pT->pP->sDT.wSt0 |=  (0x02);else
						//if ((pEV.byCause==EV_1T0_ST)&&(pEV.byAddr==0))
						//	pT->pP->sDT.wSt0 &= ~(0x02);else
					break;
					case REG_SOFTS_ADDR:
						//Активность верхнего входа
						if ((pEV.byCause==EV_0T1_CH)&&(pEV.byAddr==0))
						{
						 pT->pP->sDT.wSt0 |=  (0x01);
						 pT->pP->sDT.wParam = pT->pP->sDT.wJob0;
						} else
						if ((pEV.byCause==EV_1T0_CH)&&(pEV.byAddr==0))
						{
						 pT->pP->sDT.wSt0 &= ~(0x01);
						 pT->pP->sDT.wParam = pT->pP->sDT.wJob1;
                         if (!(pT->pP->sDT.wSt0 & 0x02)) pT->pP->sDT.wParam = 0;
						} else
						//Активность нижнего входа
						if ((pEV.byCause==EV_0T1_CH)&&(pEV.byAddr==1))
						{
					  	 pT->pP->sDT.wSt0 |=  (0x02);
						 if (!(pT->pP->sDT.wSt0 & 0x01)) pT->pP->sDT.wParam = pT->pP->sDT.wJob1;
						} else
						if ((pEV.byCause==EV_1T0_CH)&&(pEV.byAddr==1))
						{
 						 pT->pP->sDT.wSt0 &= ~(0x02);
						 if (!(pT->pP->sDT.wSt0 & 0x01)) pT->pP->sDT.wParam = 0;
						}
					break;
				 }
			break;
			default:
            break;
		   }
      break;
	  case DIR_101MD:
	  break;
	  default:
	  break;
	}
	return TRUE;
}
/*
typedef struct _tagLVData
{
UINT wParam;
}SLVDATA;
*/
PVOID CLevel_GetData(This,BYTE *pData,WORD *nLen)
{
    DECLARE_MULTI_OPEN(CLevel,CDevice)
	pB->GetWordParam(pB,(BYTE*)&pT->pP->sDT.wSt0,&pData[0]);
	pB->GetWordParam(pB,(BYTE*)&pT->pP->sDT.wJob0,&pData[2]);
	pB->GetWordParam(pB,(BYTE*)&pT->pP->sDT.wJob1,&pData[4]);
	pB->GetWordParam(pB,(BYTE*)&pT->pP->sDT.wParam,&pData[6]);
	*nLen += pB->m_nSize;if (*nLen>350) *nLen=0;
	return pData;
}
void CLevel_CLevel(This)
{
    DECLARE_MULTI_OPEN(CLevel,CDevice)
	DECLARE_VIRTUAL_FUNC(CLevel,EventHandler)
	DECLARE_VIRTUAL_FUNC(CLevel,InitTCHN)
	DECLARE_VIRTUAL_FUNC(CLevel,PreProc)
	DECLARE_VIRTUAL_FUNC(CLevel,Processing)
	DECLARE_VIRTUAL_FUNC(CLevel,PostProc)
	DECLARE_VIRTUAL_FUNC(CLevel,GetData)
}
void CLevel_DCLevel(This)
{
	DECLARE_MULTI_OPEN(CLevel,CDevice)
}
DECLARE_MULTI_CREATE(CLevel,CDevice)
```

#### bnrmeasur.h
```c
/********************************************************************
 * COPYRIGHT -- Kontora
 ********************************************************************
 * Program: bnrmain
 * File: bnraninput.h
 * Author: Abramenya
 * Created: January 19, 2009
 *******************************************************************/

#ifndef __MSMODULE_H__
#define __MSMODULE_H__
#include "typedefs.h"
#include "bnrcyclicsystem.h"
#include "bnrtu.h"
#include "bnrts.h"
#include "bnrtemper.h"
#include "bnrstgate.h"
#include "bnrpunit.h"
#include "bnrpress.h"
#include "bnrfreq.h"
#include "bnrcount.h"
#include "bnrlevel.h"
#include "bnrdevice.h"
#include "bnrdvs.h"
#include "bnrobsys.h"
//#include "bnrswitcher.h"
//#include "bnrtmcounter.h"
//#include "bnralarm.h"
#include "bnrcomputer.h"
#include "bnrflash.h"

Class CMsModule
{
	 void (*CCMsModule)(This);
	 void (*DCMsModule)(This);
Public
     void (*Init)(This,SHARDCOMPUTERTABLE *pPCTable,SSOFTSWITCHTABLE *pMsTable);
     void (*CreateChannels)(This,SDIRTABLE *pDTable);
     BOOL (*ScadaHandler)(This,SMESSAGE *pMsg);
	 BOOL (*HardControl)(This,SMESSAGE *pMsg);
	 void (*ObserveOutProc)(This);
     Virtual BOOL (*EventHandler)(This,SMESSAGE *pMsg);
     Virtual void (*CyclicProc)(This);
Public
     //SMESSAGE m_nMsg;
     CDevice **m_pDevice;
     CComputer *m_pComputer;
	 CMTimer m_nOutTMR;
	 SCONTENSTTABLE m_nST,m_nCT;
	 SHARDCOMPUTERTABLE *m_pPCT;
	 SSOFTSWITCHTABLE   *m_pPST;
	 UINT m_wAmChannel;
	 STOUTTBL mOUT;
	 //BYTE m_nSND[]
	 DECLARE_IMPLEMENT_BASE(CCyclicSystem)
}
DECLARE_DEFINITION(CMsModule)
#endif
```

#### bnrmeasur.c
```c
/********************************************************************
 * COPYRIGHT -- Kontora
 ********************************************************************
 * Program: bnrmain
 * File: bnrlsens.c
 * Author: Abramenya
 * Created: January 19, 2009
 *******************************************************************/

#include "bnrmeasur.h"
#include "bnrmain.h"
#ifdef _DEFAULT_INCLUDES
 #include <AsDefault.h>
#endif
//extern SKPPARAM nKP;
//extern SARMINTERFACE nARM0;
_GLOBAL INT nSendTmrQry;
void CMsModule_Init(This,SHARDCOMPUTERTABLE *pPCTable,SSOFTSWITCHTABLE *pMsTable)
{
    DECLARE_MULTI_OPEN(CMsModule,CCyclicSystem)
	FDEFINE(DEV_MSMDL_BOX_ID,1024);
    //InitObject(CMFlash,&pT->m_nFlash);
	//pT->m_pFlash = &pT->m_nFlash;
    pB->SetBoxID(pB,DEV_MSMDL_BOX_ID);

	InitObject(CMTimer,&pT->m_nOutTMR);
	pT->m_nOutTMR.SetTimer(&pT->m_nOutTMR,DIR_MSTOMS,DIR_MSTOMS,EV_TMR_OUT_REQ,0,0,DEV_MSMDL_BOX_ID);
	pT->m_nOutTMR.OnTimer(&pT->m_nOutTMR,10);

	//blSerialize = pT->Serialize(pT,FALSE);
	pT->CreateChannels(pT,&pMsTable->sDirectionTable[0]);

	#ifdef DEB_CMsModule
 	Info("\n(__)CKPMD::>Create Ms Module");
    #endif
	//pT->SaveInPin(pT);
}
/*
typedef struct _tagDirectionTable
{
BYTE byDirectionID;
BYTE byDirectionCode;
BYTE byAmSwitching;
BYTE byAmTI;
BYTE byAmTS;
BYTE byAmTU;
BYTE byAmTR;

  PVOID pvIn;
  PVOID pvOut;
  PVOID pSwitchTable[DEV_AMT_SWC_IDIR];
}SDIRTABLE;
typedef struct _tagTTMParams
{
BYTE byAmSlot;
BYTE byType;
STTMPARAM sTTM[4];
}STTMPARAMS;
enum _tagTeleSignal
{
TS=0,
TI,
TU,
TIS,
TC,
TPR,
TTM,
TF,
TKP,
TPU,
};
*/
void CMsModule_CreateChannels(This,SDIRTABLE *pDTable)
{
    DECLARE_MULTI_OPEN(CMsModule,CCyclicSystem)
	BYTE i,j,k=0;
	STTMPARAMS *pTT;
	PVOID pVV;
	CTu *pTU;
	CTs *pTS;
	CDevice *pD;
	CStGate *pTKP;
	CTemper *pTTM;
	CPunit  *pTPU;
	CPress  *pTPR;
	CFreq   *pTF;
	CCount  *pTC;
	CDvs    *pTVS;
	CLevel  *pLV;
	CObsSys *pOS;
	STOUTTBL mm;
	//UINT d=sizeof(STOUTTBL);
	pT->m_wAmChannel = pDTable->byAmTI;
	New(sizeof(CDevice*)*pT->m_wAmChannel,pT->m_pDevice);
	for (i=0;i<pT->m_wAmChannel;i++) pT->m_pDevice[i]=0;
	for(i=0;i<pDTable->byAmSwitching;i++)
	{
	 pTT = (STSPARAM*)pDTable->pSwitchTable[i];//Find Type
	 pVV = (PVOID)pTT;
	 switch (pTT->byType)
	 {
 	  case TKP:
 	 	 for(j=0;j<pTT->byAmSlot;j++)
		 {
		   New(sizeof(CStGate),pTKP);
		   InitObject(CStGate,pTKP);
		   pTKP->pBase->m_pComputer = pT->m_pComputer;
		   pD = pT->m_pDevice[k] = pTKP->pBase;k++;
		   pD->Init(pD,(PVOID)&((STKPARAMS*)pVV)->sTK[j]);
		 }
 	  break;
      case TC:
		 for(j=0;j<pTT->byAmSlot;j++)
		 {
		   New(sizeof(CCount),pTC);
		   InitObject(CCount,pTC);
		   pTC->pBase->m_pComputer = pT->m_pComputer;
		   pD = pT->m_pDevice[k] = pTC->pBase;k++;
		   pD->Init(pD,(PVOID)&((STCPARAMS*)pVV)->sTC[j]);
		 }
	  break;
      case TPR:
 	     for(j=0;j<pTT->byAmSlot;j++)
		 {
		   New(sizeof(CPress),pTPR);
		   InitObject(CPress,pTPR);
		   pTPR->pBase->m_pComputer = pT->m_pComputer;
		   pD = pT->m_pDevice[k] = pTPR->pBase;k++;
		   pD->Init(pD,(PVOID)&((STPRPARAMS*)pVV)->sTPR[j]);
		 }
	  break;
      case TTM:
 	     for(j=0;j<pTT->byAmSlot;j++)
		 {
		   New(sizeof(CTemper),pTTM);
		   InitObject(CTemper,pTTM);
		   pTTM->pBase->m_pComputer = pT->m_pComputer;
		   pD = pT->m_pDevice[k] = pTTM->pBase;k++;
		   pD->Init(pD,(PVOID)&((STTMPARAMS*)pVV)->sTTM[j]);
		 }
	  break;
      case TF:
 	     for(j=0;j<pTT->byAmSlot;j++)
		 {
		   New(sizeof(CFreq),pTF);
		   InitObject(CFreq,pTF);
		   pTF->pBase->m_pComputer = pT->m_pComputer;
		   pD = pT->m_pDevice[k] = pTF->pBase;k++;
		   pD->Init(pD,(PVOID)&((STFPARAMS*)pVV)->sTF[j]);
		 }
	  break;
      case TPU:
 	     for(j=0;j<pTT->byAmSlot;j++)
		 {
		   New(sizeof(CPunit),pTPU);
		   InitObject(CPunit,pTPU);
		   pTPU->pBase->m_pComputer = pT->m_pComputer;
		   pD = pT->m_pDevice[k] = pTPU->pBase;k++;
		   pD->Init(pD,(PVOID)&((SPUPARAMS*)pVV)->sTPU[j]);
		 }
	  break;
      case TU:
 	     for(j=0;j<pTT->byAmSlot;j++)
		 {
		   New(sizeof(CTu),pTU);
		   InitObject(CTu,pTU);
		   pTU->pBase->m_pComputer = pT->m_pComputer;
		   pD = pT->m_pDevice[k] = pTU->pBase;k++;
		   pD->Init(pD,(PVOID)&((STUMPARAMS*)pVV)->sTU[j]);
		 }
	  break;
      case TS:
 	     for(j=0;j<pTT->byAmSlot;j++)
		 {
		   New(sizeof(CTs),pTS);
		   InitObject(CTs,pTS);
		   pTS->pBase->m_pComputer = pT->m_pComputer;
		   pD = pT->m_pDevice[k] = pTS->pBase;k++;
		   pD->Init(pD,(PVOID)&((STSMPARAMS*)pVV)->sTS[j]);
		 }
	  break;
      case TVS:
 	     for(j=0;j<pTT->byAmSlot;j++)
		 {
		   New(sizeof(CDvs),pTVS);
		   InitObject(CDvs,pTVS);
		   pTVS->pBase->m_pComputer = pT->m_pComputer;
		   pD = pT->m_pDevice[k] = pTVS->pBase;k++;
		   pD->Init(pD,(PVOID)&((STVSPARAMS*)pVV)->sTVS[j]);
		 }
	  break;
      case TLV:
 	     for(j=0;j<pTT->byAmSlot;j++)
		 {
		   New(sizeof(CLevel),pLV);
		   InitObject(CLevel,pLV);
		   pLV->pBase->m_pComputer = pT->m_pComputer;
		   pD = pT->m_pDevice[k] = pLV->pBase;k++;
		   pD->Init(pD,(PVOID)&((SLVPARAMS*)pVV)->sLV[j]);
		 }
	  break;
      case TOS:
 	     for(j=0;j<pTT->byAmSlot;j++)
		 {
		   New(sizeof(CObsSys),pOS);
		   InitObject(CObsSys,pOS);
		   pOS->pF0  = pT->m_pDevice[20]->pChld;
		   pOS->pF1  = pT->m_pDevice[21]->pChld;
		   pOS->pF2  = pT->m_pDevice[22]->pChld;
		   pOS->pPU0 = pT->m_pDevice[27]->pChld;
		   pOS->pPU1 = pT->m_pDevice[28]->pChld;
		   pOS->pBase->m_pComputer = pT->m_pComputer;
		   pD = pT->m_pDevice[k] = pOS->pBase;k++;
		   pD->Init(pD,(PVOID)&((SOBSPARAMS*)pVV)->sOS[j]);
		 }
	  break;
	 }
     //switch(pMsg->m_sbyFor)
	}
}
BOOL CMsModule_EventHandler(This,SMESSAGE *pMsg)
{
    DECLARE_MULTI_OPEN(CMsModule,CCyclicSystem)
	CDevice *pD;
	WORD wDID;
	SINT chVS0[60],*chMS;
	REAL fVal0;
	CDvs *pVS;
	switch(pMsg->m_sbyFor)
	{
	  case DIR_MSTOMS:
		  if (pMsg->m_sbyType==EV_TMR_OUT_REQ)
		  {
			  pT->ObserveOutProc(pT);
			  pT->m_nOutTMR.OnTimer(&pT->m_nOutTMR,10);
			  //Info("\n(__)CMSMD::>EV_TMR_OUT_REQ");
		  }
		  if (pMsg->m_sbyType==EV_CHNG_PIN_REQ)
		  {
			  pT->HardControl(pT,pMsg);
		  }
	  break;
	  case DIR_OSYTOOSY:
           wDID = pMsg->m_sbySensor;
	       if (wDID<pT->m_wAmChannel)
		   {
			pD = pT->m_pDevice[wDID];
            if (pD!=0) pD->EventHandler(pD->pChld,pMsg);
		   }
	  break;
	  case DIR_PHTOMS:
		   switch(pMsg->m_sbyType)
		   {
		     case PH_VS0_REQ:
 				  pVS = pT->m_pDevice[45]->pChld;
				  strcpy((SINT*)&pVS->pP->sDT.byData[0],(SINT*)&pMsg->m_sbyInfo[0]);
 			  	  #ifdef DEB_CMsModule
				   fVal0 = atof(strcpy(chVS0,(SINT*)&pVS->pP->sDT.byData[0]));
				   printf("\n(0)VS0=%f",fVal0);
                  #endif
			 break;
		     case PH_VS1_REQ:
				  pVS = pT->m_pDevice[46]->pChld;
				  strcpy((SINT*)&pVS->pP->sDT.byData[0],(SINT*)&pMsg->m_sbyInfo[0]);
				  #ifdef DEB_CMsModule
				   fVal0 = atof(strcpy(chVS0,(SINT*)&pVS->pP->sDT.byData[0]));
 				   printf("\n(0)VS1=%f",fVal0);
				  #endif
			 break;
			 case PH_SCMD_REQ:
				  pT->ScadaHandler(pT,pMsg);
			 break;
		   }
	  break;
	  default:
	  break;
	}
	return TRUE;
}
BOOL CMsModule_ScadaHandler(This,SMESSAGE *pMsg)
{
	DECLARE_MULTI_OPEN(CMsModule,CCyclicSystem)
	CDevice *pD;
	WORD wDID;
    #ifdef DEB_CMsModule
	Info("\n(__)CMSMM::>Scada Command:%M",pMsg);
    #endif
	pB->GetWordParam(pB,&pMsg->m_sbyInfo[0],(BYTE*)&wDID);
	if (wDID<pT->m_wAmChannel)
	{
	 pD=pT->m_pDevice[wDID];
     if (pD!=0)
	 {
	  pMsg->m_sbyFor  = DIR_MSTODV;
	  pMsg->m_sbyType = PL_DATA_IND;
      pD->SEventHandler(pD,pMsg);
	 }
	}
}
BOOL CMsModule_HardControl(This,SMESSAGE *pMsg)
{
	DECLARE_MULTI_OPEN(CMsModule,CCyclicSystem)
	CDevice *pD;
	WORD wDID;
    #ifdef DEB_CMsModule
	Info("\n(__)CMSMM::>Hard Command:%M",pMsg);
    #endif
    wDID = pMsg->m_sbySensor;
	if (wDID<pT->m_wAmChannel)
	{
	 pD=pT->m_pDevice[wDID];
     if (pD!=0)
	 {
	  pMsg->m_sbyFor  = DIR_MSTODV;
      pD->EventHandler(pD->pChld,pMsg);
	 }
	}
}
void CMsModule_ObserveOutProc(This)
{
    DECLARE_MULTI_OPEN(CMsModule,CCyclicSystem)
	SMESSAGE m_sMsg;
	CDevice *pD;
    WORD i,nLen=0;
	for (i=0;i<pT->m_wAmChannel;i++)
	{
     pD = pT->m_pDevice[i];
     pD->GetData(pD->pChld,&m_sMsg.m_sbyInfo[nLen],&nLen);
	}
	m_sMsg.m_swLen        = 9+nLen;
	m_sMsg.m_sbyFrom      = DIR_MSTOTCP;
	m_sMsg.m_sbyFor       = DIR_MSTOTCP;
	m_sMsg.m_sbyIntType   = 0;
	m_sMsg.m_sbyServerID  = 0;
	m_sMsg.m_sbyType      = PL_DATA_REQ;
	m_sMsg.m_sbyDirection = 0;
	m_sMsg.m_sbySensor    = 0;
	FPUT(DEV_TCPRM_BOX_ID,(BYTE*)&m_sMsg);
    #ifdef DEB_CMsModule
	//Info("I",&m_sMsg);
	//Info("\n(__)CMSMM::>OBS::%M",&m_sMsg);
	#endif
}
_GLOBAL INT nKPC,nKPC1;
void CMsModule_CyclicProc(This)
{
    DECLARE_MULTI_OPEN(CMsModule,CCyclicSystem)
	CDevice *pD;
	WORD i;
	for (i=0;i<pT->m_wAmChannel;i++)
	{
     pD = pT->m_pDevice[i];
	 if (pD!=0)
	 pD->ObserveProc(pD);
	}
    //if (++nKPC1%20==0)pT->CheckSlot(pT);
}
void CMsModule_CMsModule(This)
{
    DECLARE_MULTI_OPEN(CMsModule,CCyclicSystem)
	DECLARE_REGISTRATION(CMsModule,Init)
	DECLARE_REGISTRATION(CMsModule,CreateChannels)
	DECLARE_REGISTRATION(CMsModule,ObserveOutProc)
	DECLARE_REGISTRATION(CMsModule,ScadaHandler)
	DECLARE_REGISTRATION(CMsModule,HardControl)
	DECLARE_VIRTUAL_FUNC(CMsModule,EventHandler)
	DECLARE_VIRTUAL_FUNC(CMsModule,CyclicProc)
}
void CMsModule_DCMsModule(This)
{
	DECLARE_MULTI_OPEN(CMsModule,CCyclicSystem)
}
DECLARE_MULTI_CREATE(CMsModule,CCyclicSystem)
```

#### bnrobsys.h
```c
/********************************************************************
 * COPYRIGHT -- Kontora
 ********************************************************************
 * Program: bnrmain
 * File: bnraninput.h
 * Author: Abramenya
 * Created: January 19, 2009
 *******************************************************************/

#ifndef __OBSYS_H__
#define __OBSYS_H__
#include "typedefs.h"
#include "bnrdevice.h"
#include "bnrpin.h"
#include "bnrcyclicsystem.h"
#include "bnrfreq.h"
#include "bnrpunit.h"
/*
//Модуль слежения
typedef struct _tagODSData
{
	//BYTE byAutoStart;
	//BYTE byPreStart;
	//BYTE byStart;
	//BYTE byStop;
	//BYTE byFinish;
    //BYTE byMode;
    DWORD dwSysState;
	WORD wJTMPreStart;
	WORD wTMPreStart;
	WORD wJTMStart;
	WORD wTMtart;
}SOBSMDATA;
*/

//Состояния модуля проливной
#define MWSY_NULL_ST00               0
#define MWSY_WAIT_OPER_ST01          1
#define MWSY_OPER_ST02               2
#define MWSY_WAIT_STOP_ST03          3
//таймеры
#define TMR_WTOP               0
#define TMR_OPER               1
#define TMR_WTST               2
//признаки
#define MS_IS_AUST          0x0001
#define MS_IS_WGHT          0x0002
#define MS_CM_AUST          0x0100
#define MS_CM_HNST          0x0200
#define MS_CM_HSTP          0x0400
#define MS_CM_FNSH          0x0800

Class CObsSys
{
	 void (*CCObsSys)(This);
	 void (*DCObsSys)(This);
Public
	 Virtual BOOL (*EventHandler)(This,SMESSAGE *pMsg);
	 Virtual void (*InitTCHN)(This,PVOID psTable);
     Virtual void (*PreProc)(This);
	 Virtual void (*Processing)(This);
     Virtual void (*PostProc)(This);
	 Virtual PVOID (*GetData)(This,BYTE *pData,WORD *nLen);
	 void (*SetMask)(This,DWORD dwMask);
	 void (*RemMask)(This,DWORD dwMask);
	 void (*StopPU)(This);
	 void (*StartPU)(This);
	 void (*StopFC)(This);
	 void (*StartFC)(This);
	 void (*StopCT)(This);
	 void (*StartCT)(This);
Protected
     BOOL (*SendMessage)(This,BYTE,BYTE);
     Virtual BOOL (*HandleTask)(This,TTask* pvTask);
	 Virtual TStateList* (*GetStateList)(This);
Public
     SOBSPARAM *pP;
     CFreq *pF0,*pF1,*pF2;
     CPunit *pPU0,*pPU1;
     BYTE m_byModuleID;
	 DECLARE_IMPLEMENT_BASE(CDevice)
}
DECLARE_DEFINITION(CObsSys)
#endif
```

#### bnrobsys.c
```c
/********************************************************************
 * COPYRIGHT -- Kontora
 ********************************************************************
 * Program: bnrmain
 * File: bnrlsens.c
 * Author: Abramenya
 * Created: January 19, 2009
 *******************************************************************/

#include "bnrobsys.h"
#include "bnrmain.h"
#ifdef _DEFAULT_INCLUDES
 #include <AsDefault.h>
#endif
_GLOBAL BYTE nFSignal;
/*
//Модуль слежения
typedef struct _tagODSData
{
	//BYTE byAutoStart;
	//BYTE byPreStart;
	//BYTE byStart;
	//BYTE byStop;
	//BYTE byFinish;
    //BYTE byMode;
    DWORD dwSysState;
	WORD wJTMPreStart;
	WORD wTMPreStart;
	WORD wJTMStart;
	WORD wTMtart;
}SOBSMDATA;
*/
char *CmpInfoSYS[]  =
{
    "==",  //JE
    "!=",  //JNE
    ">",   //JA
    "<=",  //JBE
};
char *StateInfoSYS[]  =
{
    "NULL_ST00",
	"WAIT_OPER_ST01",
	"OPER_ST02",
	"WAIT_STOP_ST03",
};
char *ValInfoSYS[]  =
{
	"FCB",
	"FCV",
	"ACD",
	"DFC",
	"MFCB",
	"MFCV",
	"CACK",
	"MCMD",
	"ISERROR",
	"ISCHNG",
	"ISCHNGTI",
	"ONE",
	"ZERO",
	"VAL0"
	"STATE",
	"STATE",
};
IMPORT_TASKCHAIN(Skip);
IMPORT_STATE(BadState);
DECLARE_TASKCHAIN(TS_EV_START_WSY_ST00)
{
	//CMD_SEND,PH_CONN_IND,DIR_101TOKP,
	CMD_START_FC,
	//CMD_SETVALUE,ACD,0,
	CMD_TIMERON,TMR_WTOP,
	CMD_SETSTATE,MWSY_WAIT_OPER_ST01,
	EXIT_D,
};
DECLARE_TASKCHAIN(TS_EV_HAND_STOP_WSY_ST00)
{
	CMD_STOP_FC,
	CMD_STOP_PU,
	CMD_STOP_CT,
	CMD_TIMEROFF,TMR_WTOP,
	CMD_TIMEROFF,TMR_OPER,
	CMD_TIMEROFF,TMR_WTST,
	CMD_SETSTATE,MWSY_NULL_ST00,
	EXIT_D,
};
//ST_01///////////////////////////////////////
DECLARE_TASKCHAIN(TS_EV_TMR_WTOP_ST01)
{
	CMD_START_PU,
	CMD_START_CT,
	CMD_TIMERON,TMR_OPER,
	CMD_SETSTATE,MWSY_OPER_ST02,
	EXIT_D,
};
//ST_02///////////////////////////////////////
DECLARE_TASKCHAIN(TS_EV_TMR_OPER_ST02)
{
	CMD_STOP_PU,
	CMD_TIMERON,TMR_WTST,
    CMD_SETSTATE,MWSY_WAIT_STOP_ST03,
	EXIT_D,
};
DECLARE_TASKCHAIN(TS_EV_CT_OFF_ST02)
{
	CMD_STOP_CT,
	CMD_STOP_PU,
	CMD_STOP_FC,
	CMD_TIMERON,TMR_WTST,
	CMD_SETSTATE,MWSY_WAIT_STOP_ST03,
	EXIT_D,
};
//ST_03///////////////////////////////////////
DECLARE_TASKCHAIN(TS_EV_TMR_WTST_ST03)
{
	CMD_STOP_FC,
	CMD_SETSTATE,MWSY_NULL_ST00,
	EXIT_D,
};
DECLARE_STATE(ST_MWSY_NULL_ST00)
{
	{ EV_START_WSY_REQ,         TS_EV_START_WSY_ST00 },
	{ EV_HAND_START_WSY_REQ,    TS_EV_TMR_WTOP_ST01 },
	{ EV_HAND_STOP_WSY_REQ,     TS_EV_HAND_STOP_WSY_ST00 },
    { EV_UNKNOWN_REQ,           Skip               }
};
DECLARE_STATE(ST_MWSY_WAIT_OPER_ST01)
{
    { EV_TMR_WTOP_REQ,          TS_EV_TMR_WTOP_ST01  },
	{ EV_HAND_STOP_WSY_REQ,     TS_EV_HAND_STOP_WSY_ST00 },
    { EV_UNKNOWN_REQ,           Skip               }
};
DECLARE_STATE(ST_MWSY_OPER_ST02)
{
    { EV_TMR_OPER_REQ,          TS_EV_TMR_OPER_ST02  },
    { EV_CT_OFF_REQ,            TS_EV_CT_OFF_ST02  },
	{ EV_HAND_STOP_WSY_REQ,     TS_EV_HAND_STOP_WSY_ST00 },
    { EV_UNKNOWN_REQ,           Skip               }
};
DECLARE_STATE(ST_MWSY_WAIT_STOP_ST03)
{
    { EV_TMR_WTST_REQ,          TS_EV_TMR_WTST_ST03  },
	{ EV_HAND_STOP_WSY_REQ,     TS_EV_HAND_STOP_WSY_ST00 },
    { EV_UNKNOWN_REQ,           Skip               }
};
DECLARE_STATELIST(STL_OSY_PROT)
{
    { MWSY_NULL_ST00,           ST_MWSY_NULL_ST00 },
	{ MWSY_WAIT_OPER_ST01,      ST_MWSY_WAIT_OPER_ST01 },
	{ MWSY_OPER_ST02,           ST_MWSY_OPER_ST02 },
	{ MWSY_WAIT_STOP_ST03,      ST_MWSY_WAIT_STOP_ST03 },
    { S_BAD,                    BadState       }
};
_GLOBAL WORD wglValue;
BOOL CObsSys_HandleTask(This,TTask* pTask)
{
    DECLARE_MULTI_OPEN(CObsSys,CDevice)
	BYTE V0,V1,V2,SIGN,LBL;
	BOOL byLoop;
	BYTE *p_EvArr = pTask;
	INT nBTI,nBTS;
	//STISTAG sTS;
	for(;*pTask!=EXIT_D;pTask++)
	//while(*pTask!=EXIT_D)
    {
	  switch (*pTask)
	  {
         case CMD_INCC:
			  pB->v[*(++pTask)]++;
			  pB->v[*pTask] &= 0x01;
              #ifdef DEB_CObsSys
			  Info("\n(%b)COBSY::>INCC::%s=%b",&pT->m_byModuleID,ValInfoSYS[*pTask],&pB->v[*pTask]);
              #endif
		 break;
	  	 case CMD_SETSTATE:
			  V1 = *(++pTask);
			  //if(*pTask==STATE_101) V1 = pB->v[STATE_101];
			  pB->SetState(pB,V1);
              #ifdef DEB_CObsSys
			  Info("\n(%b)COBSY::>STAT::%s->%s ",&pT->m_byModuleID,StateInfoSYS[pB->v[STATE_WSY]],StateInfoSYS[V1]);
			  //Info("\n(%b)CWSYS[%b]::>STAT:/--------New--------/",&pT->m_bySystemID,&pT->m_bySensorID);
              #endif
			  pB->v[STATE_WSY] = V1;
         break;
		 case CMD_SEND:
			  V0 = *(++pTask);
			  V1 = *(++pTask);
			  //pT->SendMessage(pT,V0,V1);
              #ifdef DEB_CObsSys
			  Info("\n(%b)COBSY::>SEND::[%b][%b]",&pT->m_byModuleID,&V0,&V1);
              #endif
		 break;
		 case CMD_SETVALUE:
			  V0 = *(++pTask);
			  pB->v[V0] = *(++pTask);
              #ifdef DEB_CObsSys
			  Info("\n(%b)COBSY::>SETV::%s=%b",&pT->m_byModuleID,ValInfoSYS[V0],&pB->v[V0]);
              #endif
		 break;
		 case CMD_MOV:
			  V1 = *(++pTask);
			  pB->v[V1] = pB->v[*(++pTask)];
              #ifdef DEB_CObsSys
			  Info("\n(%b)COBSY::>MOVV::%s<-%s",&pT->m_byModuleID,ValInfoSYS[*(pTask-1)],ValInfoSYS[*pTask]);
              #endif
		 break;
		 case CMD_CMP:
			  byLoop=1;
			  V1 = pB->v[*(++pTask)];
			  SIGN = *(++pTask);
			  V2 = pB->v[*(++pTask)];
			  LBL = *(++pTask);
              switch(SIGN)
              {
                case JE:
                if (V1==V2) byLoop=0; else byLoop= 1;
                break;
                case JNE:
                if (V1!=V2) byLoop=0; else byLoop=-1;
                break;
                case JA:
                if (V1>V2)  byLoop=0; else byLoop= 1;
                break;
                case JBE:
                if (V1<=V2) byLoop=0; else byLoop=-1;
                break;
                default:
                break;
               }
               #ifdef DEB_CObsSys
               Info("\n(%b)COBSY::>CMPV::%s%s%s",&pT->m_byModuleID,ValInfoSYS[*(pTask-3)],CmpInfoSYS[SIGN+byLoop],ValInfoSYS[*(pTask-1)]);
               #endif
               if(byLoop==0) pTask = p_EvArr+LBL-1;
		 break;
		 case CMD_TIMERON:
			  V0 = *(++pTask);//Timer ID
			  //V1 = *(++pTask);//Time
			  pB->m_nATmr[V0].OnTimer(&pB->m_nATmr[V0],pB->m_dwTM[V0]);
              #ifdef DEB_CObsSys
			  Info("\n(%b)COBSY::>TMON::[%b][%b]",&pT->m_byModuleID,&V0,&pB->m_dwTM[V0]);
	          #endif
		 break;
		 case CMD_TIMEROFF:
			  V0 = *(++pTask);
			  pB->m_nATmr[V0].OfTimer(&pB->m_nATmr[V0]);
              #ifdef DEB_CObsSys
			  Info("\n(%b)COBSY::>TMOF::[%b]",&pT->m_byModuleID,&V0);
              #endif
		 break;
		 case CMD_STOP_FC:
			  pT->StopFC(pT);
              #ifdef DEB_CObsSys
			  Info("\n(%b)COBSY::>STOP_FC",&pT->m_byModuleID);
              #endif
		 break;
		 case CMD_START_FC:
			  pT->StartFC(pT);
              #ifdef DEB_CObsSys
			  Info("\n(%b)COBSY::>START_FC",&pT->m_byModuleID);
              #endif
		 break;
		 case CMD_STOP_PU:
			  pT->StopPU(pT);
              #ifdef DEB_CObsSys
			  Info("\n(%b)COBSY::>STOP_PU",&pT->m_byModuleID);
              #endif
		 break;
		 case CMD_START_PU:
			  pT->StartPU(pT);
              #ifdef DEB_CObsSys
			  Info("\n(%b)COBSY::>START_PU",&pT->m_byModuleID);
              #endif
		 break;
		 case CMD_STOP_CT:
			  pT->StopCT(pT);
              #ifdef DEB_CObsSys
			  Info("\n(%b)COBSY::>STOP_CT",&pT->m_byModuleID);
              #endif
		 break;
		 case CMD_START_CT:
			  pT->StartCT(pT);
              #ifdef DEB_CObsSys
			  Info("\n(%b)COBSY::>START_CT",&pT->m_byModuleID);
              #endif
		 break;
		 default:
		 break;
	  };
	}
	return TRUE;
}
/*
//Модуль слежения
typedef struct _tagODSData
{
	//BYTE byAutoStart;
	//BYTE byPreStart;
	//BYTE byStart;
	//BYTE byStop;
	//BYTE byFinish;
    //BYTE byMode;
    DWORD dwSysState;
	WORD wJTMPreStart;
	WORD wTMPreStart;
	WORD wJTMStart;
	WORD wTMStart;
	WORD wJTMWait;
	WORD wTMWait;
}SOBSMDATA;
/*
//Состояния модуля проливной
#define MWSY_NULL_ST00               0
#define MWSY_WAIT_OPER_ST01          1
#define MWSY_OPER_ST02               2
#define MWSY_WAIT_STOP_ST03          3

  //Сообщения пролива
#define EV_START_WSY_REQ             _KPMOD_SHIFT + 76 //Запуск модуля
#define EV_HAND_STOP_WSY_REQ         _KPMOD_SHIFT + 77 //Ручной останов
#define EV_HAND_START_WSY_REQ        _KPMOD_SHIFT + 78 //Ручной старт
#define EV_TMR_WTOP_REQ              _KPMOD_SHIFT + 79 //Таймер Ожидания Операционного режима
#define EV_TMR_OPER_REQ              _KPMOD_SHIFT + 80 //Таймер Операционного режима
#define EV_TMR_WTST_REQ              _KPMOD_SHIFT + 81 //Таймер Ожидания Успокоения Жидкости
*/
void CObsSys_InitTCHN(This,PVOID psTable)
{
    DECLARE_MULTI_OPEN(CObsSys,CDevice)
	CSlot *pSL;
	CComputer *pCM = pB->m_pComputer;
	pT->pP = (SOBSPARAM*)psTable;
	pB->m_nSize = sizeof(DWORD)+6*sizeof(WORD);

	pB->m_pStateList  = STL_OSY_PROT;
    pB->m_byAutoState = MWSY_NULL_ST00;
	pB->SetState(pB,MWSY_NULL_ST00);
	InitObject(CMTimer,&pB->m_nATmr[TMR_WTOP]);
	InitObject(CMTimer,&pB->m_nATmr[TMR_OPER]);
	InitObject(CMTimer,&pB->m_nATmr[TMR_WTST]);
	pT->m_byModuleID  = pT->pP->byID;
	pB->v[STATE_WSY]  = MWSY_NULL_ST00;
    //void (*SetTimer)(This,BYTE byFor,BYTE byFrom,BYTE byEvent,BYTE byDir,BYTE bySens,BYTE byBox);

	pB->m_nATmr[TMR_WTOP].SetTimer(&pB->m_nATmr[TMR_WTOP],DIR_OSYTOOSY,DIR_OSYTOOSY,EV_TMR_WTOP_REQ,0,pT->pP->byID,DEV_MSMDL_BOX_ID);
	pB->m_dwTM[TMR_WTOP] = 10*pT->pP->sDT.wJTMPreStart;

	pB->m_nATmr[TMR_OPER].SetTimer(&pB->m_nATmr[TMR_OPER],DIR_OSYTOOSY,DIR_OSYTOOSY,EV_TMR_OPER_REQ,0,pT->pP->byID,DEV_MSMDL_BOX_ID);
	pB->m_dwTM[TMR_OPER] = 10*pT->pP->sDT.wJTMStart;

	pB->m_nATmr[TMR_WTST].SetTimer(&pB->m_nATmr[TMR_WTST],DIR_OSYTOOSY,DIR_OSYTOOSY,EV_TMR_WTST_REQ,0,pT->pP->byID,DEV_MSMDL_BOX_ID);
	pB->m_dwTM[TMR_WTST] = 10*pT->pP->sDT.wJTMWait;

	//pB->HandleEvent(pB,pMsg->m_sbyType);
    #ifdef DEB_CObsSys
	//Info("\n(%b)CTLSG::>Create TeleSignal.",&pB->m_byID);
    #endif
}
TStateList* CObsSys_GetStateList(This)
{
    DECLARE_MULTI_OPEN(CObsSys,CDevice)
	return pB->m_pStateList;
}
void CObsSys_PreProc(This)
{
    DECLARE_MULTI_OPEN(CObsSys,CDevice)
}
_GLOBAL INT nTSCH;
void CObsSys_Processing(This)
{
	DECLARE_MULTI_OPEN(CObsSys,CDevice)
}
void CObsSys_PostProc(This)
{
	DECLARE_MULTI_OPEN(CObsSys,CDevice)
}
BOOL CObsSys_EventHandler(This,SMESSAGE *pMsg)
{
    DECLARE_MULTI_OPEN(CObsSys,CDevice)
    #ifdef DEB_CObsSys
	Info("\n(%b)CTLSG::>INPT::%M",&pB->m_nCD.wDeviceID,pMsg);
    #endif
	switch(pMsg->m_sbyFor)
	{
	  case DIR_MSTODV:
		   switch(pMsg->m_sbyType)
		   {
		    case PL_DATA_IND:
                 switch(pB->m_nCD.byParam0)
				 {
				   case CTR_TR:
                        switch (pB->m_nCD.byParam1)
					    {
						  case 0:
							   pT->pP->sDT.wJTMPreStart = (WORD)(pB->m_nCD.fParam0);
							   pB->m_dwTM[TMR_WTOP] = 10*pT->pP->sDT.wJTMPreStart;
						  break;
						  case 1:
							   pT->pP->sDT.wJTMStart = (WORD)(pB->m_nCD.fParam0);
							   pB->m_dwTM[TMR_OPER] = 10*pT->pP->sDT.wJTMStart;
						  break;
						  case 2:
							   pT->pP->sDT.wJTMWait = (WORD)(pB->m_nCD.fParam0);
							   pB->m_dwTM[TMR_WTST] = 10*pT->pP->sDT.wJTMWait;
						  break;
						  default:
						  break;
					    }
				   break;
                   case CTR_TU:
                         switch (pB->m_nCD.byParam1)
					    {
						  case 0:
							   if (pB->m_nCD.wParam0==0) pT->RemMask(pT,MS_IS_AUST);else  //Признак Автостарта
							   if (pB->m_nCD.wParam0==1) pT->SetMask(pT,MS_IS_AUST);      //Признак Автостарта
						  break;
						  case 1:
							   //Признак работы на весы
							   if (pB->m_nCD.wParam0==0)
							   {
								pT->RemMask(pT,MS_IS_WGHT);
                                pT->pPU0->ClosePU(pT->pPU0);
                                pT->pPU1->ClosePU(pT->pPU1);
							   }
							   if (pB->m_nCD.wParam0==1) pT->SetMask(pT,MS_IS_WGHT);//Признак работы на весы
						  break;
						  case 2:
							   if (pB->m_nCD.wParam0==1) pT->SetMask(pT,MS_CM_AUST);//Автостарт с продувкой
							   pT->RemMask(pT,MS_CM_HSTP);
							   pT->RemMask(pT,MS_CM_FNSH);
							   if (pT->pP->sDT.wSt0 & MS_IS_AUST)    pB->HandleEvent(pB,EV_START_WSY_REQ); else
							   if (!(pT->pP->sDT.wSt0 & MS_IS_AUST)) pT->StartFC(pT);
						  break;
						  case 3:
							   if (!(pT->pP->sDT.wSt0 & MS_CM_AUST)) break;
							   if (pB->m_nCD.wParam0==1) pT->SetMask(pT,MS_CM_HNST);//Ручной Старт начала счета
							   if (!(pT->pP->sDT.wSt0 & MS_IS_AUST))
							   {
								 pT->RemMask(pT,MS_CM_AUST);
								 pB->HandleEvent(pB,EV_HAND_START_WSY_REQ);
							   }
							   pT->RemMask(pT,MS_CM_HSTP);
						  break;
						  case 4:
							   if (pB->m_nCD.wParam0==1) pT->SetMask(pT,MS_CM_HSTP);//Ручной Стоп установки с АРМ
							   pT->RemMask(pT,MS_CM_AUST);
							   pT->RemMask(pT,MS_CM_HNST);
							   pT->RemMask(pT,MS_CM_FNSH);
							   pB->HandleEvent(pB,EV_HAND_STOP_WSY_REQ);
						  break;
  					      default:
						  break;
					    }
				   break;
				   default:
				   break;
				 }
		    break;
			default:
			 //pB->HandleEvent(pB,pMsg->m_sbyType);
            break;
		   }
      break;
	  case DIR_OSYTOOSY:
		   switch (pMsg->m_sbyType)
		   {
		    case EV_TMR_WTOP_REQ:
				 pT->RemMask(pT,MS_CM_AUST);
				 pT->SetMask(pT,MS_CM_HNST);
			break;
		    case EV_TMR_OPER_REQ:
				 pT->RemMask(pT,MS_CM_AUST);
			break;
		    case EV_TMR_WTST_REQ:
				 pT->RemMask(pT,MS_CM_AUST);
				 pT->RemMask(pT,MS_CM_HNST);
				 pT->SetMask(pT,MS_CM_FNSH);
			break;
		   }
           pB->HandleEvent(pB,pMsg->m_sbyType);
	  break;
	  default:
	  break;
	}
	return TRUE;
}
/*
//Модуль слежения
typedef struct _tagODSData
{
	//BYTE byAutoStart;
	//BYTE byPreStart;
	//BYTE byStart;
	//BYTE byStop;
	//BYTE byFinish;
    //BYTE byMode;
    DWORD dwSysState;
	WORD wJTMPreStart;
	WORD wTMPreStart;
	WORD wJTMStart;
	WORD wTMStart;
	WORD wJTMWait;
	WORD wTMWait;
}SOBSMDATA;
*/
void CObsSys_StopPU(This)
{
    DECLARE_MULTI_OPEN(CObsSys,CDevice)
	if (pT->pP->sDT.wSt0 & MS_IS_WGHT)
	{
	 pT->pPU0->StopPU(pT->pPU0);
     pT->pPU1->StopPU(pT->pPU1);
	}
}
void CObsSys_StartPU(This)
{
    DECLARE_MULTI_OPEN(CObsSys,CDevice)
	if (pT->pP->sDT.wSt0 & MS_IS_WGHT)
	{
	 pT->pPU0->StartPU(pT->pPU0);
     pT->pPU1->StartPU(pT->pPU1);
	}
}
void CObsSys_StopFC(This)
{
    DECLARE_MULTI_OPEN(CObsSys,CDevice)
	pT->pF0->StopFC(pT->pF0);
	pT->pF1->StopFC(pT->pF1);
	pT->pF2->StopFC(pT->pF2);
}
void CObsSys_StartFC(This)
{
    DECLARE_MULTI_OPEN(CObsSys,CDevice)
	pT->pF0->StartFC(pT->pF0);
	pT->pF1->StartFC(pT->pF1);
	pT->pF2->StartFC(pT->pF2);
}
void CObsSys_SetMask(This,DWORD dwMask)
{
    DECLARE_MULTI_OPEN(CObsSys,CDevice)
	pT->pP->sDT.wSt0 |= dwMask;
}
void CObsSys_RemMask(This,DWORD dwMask)
{
    DECLARE_MULTI_OPEN(CObsSys,CDevice)
	pT->pP->sDT.wSt0 &= ~dwMask;
}
void CObsSys_StopCT(This)
{
    DECLARE_MULTI_OPEN(CObsSys,CDevice)

}
void CObsSys_StartCT(This)
{
    DECLARE_MULTI_OPEN(CObsSys,CDevice)

}

BOOL CObsSys_SendMessage(This,BYTE byMsgType,BYTE byFor)
{
    DECLARE_MULTI_OPEN(CObsSys,CDevice)
	switch(byFor)
	{
	  case DIR_101TOPH:
		   switch(byMsgType)
		   {
		     case PH_DATA1_RES:

			 break;
		   }
	  break;
	}
    return TRUE;
}
PVOID CObsSys_GetData(This,BYTE *pData,WORD *nLen)
{
    DECLARE_MULTI_OPEN(CObsSys,CDevice)
	pT->pP->sDT.wTMPreStart = (WORD)(pB->m_nATmr[TMR_WTOP].GetTime(&pB->m_nATmr[TMR_WTOP])/10);
    pT->pP->sDT.wTMStart    = (WORD)(pB->m_nATmr[TMR_OPER].GetTime(&pB->m_nATmr[TMR_OPER])/10);
    pT->pP->sDT.wTMWait     = (WORD)(pB->m_nATmr[TMR_WTST].GetTime(&pB->m_nATmr[TMR_WTST])/10);
	pB->GetDWordParam(pB,(BYTE*)&pT->pP->sDT.wSt0,&pData[0]);
	pB->GetWordParam(pB,(BYTE*)&pT->pP->sDT.wJTMPreStart,&pData[4]);
	pB->GetWordParam(pB,(BYTE*)&pT->pP->sDT.wTMPreStart,&pData[6]);
	pB->GetWordParam(pB,(BYTE*)&pT->pP->sDT.wJTMStart,&pData[8]);
	pB->GetWordParam(pB,(BYTE*)&pT->pP->sDT.wTMStart,&pData[10]);
	pB->GetWordParam(pB,(BYTE*)&pT->pP->sDT.wJTMWait,&pData[12]);
	pB->GetWordParam(pB,(BYTE*)&pT->pP->sDT.wTMWait,&pData[14]);
	*nLen += pB->m_nSize;if (*nLen>350) *nLen=0;
	return pData;
}
void CObsSys_CObsSys(This)
{
    DECLARE_MULTI_OPEN(CObsSys,CDevice)
	DECLARE_REGISTRATION(CObsSys,SendMessage)
	DECLARE_REGISTRATION(CObsSys,StopPU)
	DECLARE_REGISTRATION(CObsSys,StartPU)
	DECLARE_REGISTRATION(CObsSys,StopFC)
	DECLARE_REGISTRATION(CObsSys,StartFC)
	DECLARE_REGISTRATION(CObsSys,StopCT)
	DECLARE_REGISTRATION(CObsSys,StartCT)
	DECLARE_REGISTRATION(CObsSys,SetMask)
	DECLARE_REGISTRATION(CObsSys,RemMask)
	DECLARE_VIRTUAL_FUNC(CObsSys,EventHandler)
	DECLARE_VIRTUAL_FUNC(CObsSys,InitTCHN)
	DECLARE_VIRTUAL_FUNC(CObsSys,PreProc)
	DECLARE_VIRTUAL_FUNC(CObsSys,Processing)
	DECLARE_VIRTUAL_FUNC(CObsSys,PostProc)
	DECLARE_VIRTUAL_FUNC(CObsSys,GetData)
	DECLARE_VIRTUAL_FUNC(CObsSys,HandleTask)
	DECLARE_VIRTUAL_FUNC(CObsSys,GetStateList)
}
void CObsSys_DCObsSys(This)
{
	DECLARE_MULTI_OPEN(CObsSys,CDevice)
}
DECLARE_MULTI_CREATE(CObsSys,CDevice)
```

#### bnrpress.h
```c
/********************************************************************
 * COPYRIGHT -- Kontora
 ********************************************************************
 * Program: bnrmain
 * File: bnraninput.h
 * Author: Abramenya
 * Created: January 19, 2009
 *******************************************************************/

#ifndef __PRESS_H__
#define __PRESS_H__
#include "typedefs.h"
#include "bnrdevice.h"
#include "bnrpin.h"

Class CPress
{
	 void (*CCPress)(This);
	 void (*DCPress)(This);
Public
     BYTE (*CheckTS)(This);
	 Virtual BOOL (*EventHandler)(This,SMESSAGE *pMsg);
	 Virtual void (*InitTCHN)(This,PVOID psTable);
     Virtual void (*PreProc)(This);
	 Virtual void (*Processing)(This);
     Virtual void (*PostProc)(This);
	 Virtual void (*SetInPinEvent)(This);
	 Virtual void (*SaveAlarmPin)(This);
	 Virtual void (*SendObsrveMsg)(This);
	 Virtual PVOID (*GetData)(This,BYTE *pData,WORD *nLen);
Public
     STPRPARAM *pP;
	 WORD *m_pwVL0;
	 DECLARE_IMPLEMENT_BASE(CDevice)
}
DECLARE_DEFINITION(CPress)
#endif
```

#### bnrpress.c
```c
/********************************************************************
 * COPYRIGHT -- Kontora
 ********************************************************************
 * Program: bnrmain
 * File: bnrlsens.c
 * Author: Abramenya
 * Created: January 19, 2009
 *******************************************************************/

#include "bnrpress.h"
#include "bnrmain.h"
#ifdef _DEFAULT_INCLUDES
 #include <AsDefault.h>
#endif
_GLOBAL BYTE nFSignal;
void CPress_InitTCHN(This,PVOID psTable)
{
    DECLARE_MULTI_OPEN(CPress,CDevice)
	CSlot *pSL;
	CPin *m_pPN0;
	BOOL *m_pbVL0;
	CComputer *pCM = pB->m_pComputer;

	pT->pP = (STPRPARAM*)psTable;
	pB->m_nSize = 2*sizeof(WORD);

	pSL          = pCM->GetSlot(pCM,pT->pP->bySlot);
	m_pPN0       = pSL->GetPin(pSL->pChld,pT->pP->byPin);
    pT->m_pwVL0 = (WORD*)m_pPN0->GetAddrPin(m_pPN0->pChld);

    #ifdef DEB_CPress
	//Info("\n(%b)CTLSG::>Create TeleSignal.",&pB->m_byID);
    #endif
}
void CPress_PreProc(This)
{
    DECLARE_MULTI_OPEN(CPress,CDevice)
	pT->pP->sDT.wParam = *pT->m_pwVL0;
}
_GLOBAL INT nTSCH;
void CPress_Processing(This)
{
	DECLARE_MULTI_OPEN(CPress,CDevice)
}
void CPress_PostProc(This)
{
	DECLARE_MULTI_OPEN(CPress,CDevice)
}
BYTE CPress_CheckTS(This)
{
    DECLARE_MULTI_OPEN(CPress,CDevice)
    //return pB->m_pPN->GetState(pB->m_pPN);
	return 0;
}
BOOL CPress_EventHandler(This,SMESSAGE *pMsg)
{
    DECLARE_MULTI_OPEN(CPress,CDevice)
    BYTE byID = pMsg->m_sbySensor;
	BYTE byParamType = pMsg->m_sbyInfo[3];
    #ifdef DEB_CPress
	Info("\n(%b)CTLSG::>INPT::%M",&pB->m_byID,pMsg);
    #endif
	switch(pMsg->m_sbyFor)
	{
	  case DIR_101TOKP:
		   switch(pMsg->m_sbyType)
		   {
		    case PL_DATA_IND:
				 //Info("\n(%b)CTLSG::>DL_DATA_IND::>%M",&pB->m_byID,pMsg);
				 switch(byParamType)
				 {
				   case EN_SET_PERIOD:
					    //pT->m_byCSetPulce = pMsg->m_sbyInfo[3];
					    //pT->m_bySetPulce  = pT->m_byCSetPulce;
				   break;
				   case EN_REM_PERIOD:
					    //pT->m_byRemPulce  = pMsg->m_sbyInfo[3];
						//pT->m_byCRemPulce = pT->m_byRemPulce;
				   break;
				   case EN_PIN_ALMODE:
                        //pT->m_byAlarmMode = pMsg->m_sbyInfo[3];
				   break;
				   default:
				   break;
				 }
		    break;
			default:
            break;
		   }
      break;
	  case DIR_101MD:
	  break;
	  default:
	  break;
	}
	return TRUE;
}
void CPress_SetInPinEvent(This)
{
    DECLARE_MULTI_OPEN(CPress,CDevice)
}
void CPress_SaveAlarmPin(This)
{
	DECLARE_MULTI_OPEN(CPress,CDevice)
}
void CPress_SendObsrveMsg(This)
{
    DECLARE_MULTI_OPEN(CPress,CDevice)
}
/*
typedef struct _tagTPRData
{
UINT wJob;
UINT wParam;
}SPRMDATA;
*/
PVOID CPress_GetData(This,BYTE *pData,WORD *nLen)
{
    DECLARE_MULTI_OPEN(CPress,CDevice)
    pB->GetWordParam(pB,(BYTE*)&pT->pP->sDT.wJob,&pData[0]);
	pB->GetWordParam(pB,(BYTE*)&pT->pP->sDT.wParam,&pData[2]);
	*nLen += pB->m_nSize;if (*nLen>350) *nLen=0;
	return pData;
}
void CPress_CPress(This)
{
    DECLARE_MULTI_OPEN(CPress,CDevice)
	DECLARE_REGISTRATION(CPress,CheckTS)
	DECLARE_VIRTUAL_FUNC(CPress,EventHandler)
	DECLARE_VIRTUAL_FUNC(CPress,InitTCHN)
	DECLARE_VIRTUAL_FUNC(CPress,PreProc)
	DECLARE_VIRTUAL_FUNC(CPress,Processing)
	DECLARE_VIRTUAL_FUNC(CPress,PostProc)
	DECLARE_VIRTUAL_FUNC(CPress,SetInPinEvent)
	DECLARE_VIRTUAL_FUNC(CPress,SaveAlarmPin)
	DECLARE_VIRTUAL_FUNC(CPress,SendObsrveMsg)
	DECLARE_VIRTUAL_FUNC(CPress,GetData)
}
void CPress_DCPress(This)
{
	DECLARE_MULTI_OPEN(CPress,CDevice)
}
DECLARE_MULTI_CREATE(CPress,CDevice)
```

#### bnrpunit.h
```c
/********************************************************************
 * COPYRIGHT -- Kontora
 ********************************************************************
 * Program: bnrmain
 * File: bnraninput.h
 * Author: Abramenya
 * Created: January 19, 2009
 *******************************************************************/

#ifndef __TPUNIT_H__
#define __TPUNIT_H__
#include "typedefs.h"
#include "bnrdevice.h"
#include "bnrpin.h"
#include "bnrdevtu.h"
#include "bnrdevts.h"
Class CPunit
{
	 void (*CCPunit)(This);
	 void (*DCPunit)(This);
Public
     void (*StartPU)(This);
     void (*StopPU)(This);
     void (*ClosePU)(This);
	 Virtual BOOL (*EventHandler)(This,SMESSAGE *pMsg);
	 Virtual void (*InitTCHN)(This,PVOID psTable);
     Virtual void (*PreProc)(This);
	 Virtual void (*Processing)(This);
     Virtual void (*PostProc)(This);
	 Virtual PVOID (*GetData)(This,BYTE *pData,WORD *nLen);
Public
     SPUPARAM *pP;
	 CDevTU *pTU0;
     CDevTS *pTS0;
     CDevTS *pTS1;
     CDevTS *pTS2;
	 DECLARE_IMPLEMENT_BASE(CDevice)
}
DECLARE_DEFINITION(CPunit)
#endif
```

#### bnrpunit.c
```c
/********************************************************************
 * COPYRIGHT -- Kontora
 ********************************************************************
 * Program: bnrmain
 * File: bnrlsens.c
 * Author: Abramenya
 * Created: January 19, 2009
 *******************************************************************/

#include "bnrpunit.h"
#include "bnrmain.h"
#ifdef _DEFAULT_INCLUDES
 #include <AsDefault.h>
#endif
_GLOBAL BYTE nFSignal;
void CPunit_InitTCHN(This,PVOID psTable)
{
    DECLARE_MULTI_OPEN(CPunit,CDevice)
	CSlot *pSL;
	CPin *m_pPN0;
	BOOL *m_pbVL0;
	BOOL *m_pbAVL0;
	CComputer *pCM = pB->m_pComputer;
	pT->pP = (SPUPARAM*)psTable;
	pB->m_nSize = 3*sizeof(WORD);

	//Выход открытия
	pSL          = pCM->GetSlot(pCM,pT->pP->bySlot);
	m_pPN0       = pSL->GetPin(pSL->pChld,pT->pP->byPin);
    m_pbVL0 = (BOOL*)m_pPN0->GetAddrPin(m_pPN0->pChld);
	New(sizeof(CDevTU),pT->pTU0);
	InitObject(CDevTU,pT->pTU0);
    pT->pTU0->Init(pT->pTU0,m_pbVL0,pT->pP->byID,0,EN_OPEN,EN_DIRECT,10);
	pT->pTU0->SetTU(pT->pTU0,DEV_MSMDL_BOX_ID,DIR_MSTOMS,EV_CHNG_PIN_REQ);

	//Вход левое положение
	pSL          = pCM->GetSlot(pCM,pT->pP->bySlot1);
	m_pPN0       = pSL->GetPin(pSL->pChld,pT->pP->byPin1);
    m_pbAVL0 = (BOOL*)m_pPN0->GetAddrPin(m_pPN0->pChld);
	New(sizeof(CDevTS),pT->pTS0);
	InitObject(CDevTS,pT->pTS0);
    pT->pTS0->Init(pT->pTS0,m_pPN0, m_pbAVL0,pT->pP->byID,0,EN_OPEN,PRI_HI,3,3,EN_AL_TO_AL);
	pT->pTS0->SetTS(pT->pTS0,DEV_MSMDL_BOX_ID,DIR_MSTOMS,EV_CHNG_PIN_REQ);

	//Вход среднее положение
	pSL          = pCM->GetSlot(pCM,pT->pP->bySlot2);
	m_pPN0       = pSL->GetPin(pSL->pChld,pT->pP->byPin2);
    m_pbAVL0 = (BOOL*)m_pPN0->GetAddrPin(m_pPN0->pChld);
	New(sizeof(CDevTS),pT->pTS1);
	InitObject(CDevTS,pT->pTS1);
    pT->pTS1->Init(pT->pTS1,m_pPN0, m_pbAVL0,pT->pP->byID,1,EN_OPEN,PRI_HI,3,3,EN_AL_TO_AL);
	pT->pTS1->SetTS(pT->pTS1,DEV_MSMDL_BOX_ID,DIR_MSTOMS,EV_CHNG_PIN_REQ);

	//Вход правое положение
	pSL          = pCM->GetSlot(pCM,pT->pP->bySlot3);
	m_pPN0       = pSL->GetPin(pSL->pChld,pT->pP->byPin3);
    m_pbAVL0 = (BOOL*)m_pPN0->GetAddrPin(m_pPN0->pChld);
	New(sizeof(CDevTS),pT->pTS2);
	InitObject(CDevTS,pT->pTS2);
    pT->pTS2->Init(pT->pTS2,m_pPN0, m_pbAVL0,pT->pP->byID,2,EN_OPEN,PRI_HI,3,3,EN_AL_TO_AL);
	pT->pTS2->SetTS(pT->pTS2,DEV_MSMDL_BOX_ID,DIR_MSTOMS,EV_CHNG_PIN_REQ);

    #ifdef DEB_CPunit
	//Info("\n(%b)CTLSG::>Create TeleSignal.",&pB->m_byID);
    #endif
}
void CPunit_PreProc(This)
{
    DECLARE_MULTI_OPEN(CPunit,CDevice)
	pT->pTU0->Run(pT->pTU0);
	pT->pTS0->Run(pT->pTS0);
	pT->pTS1->Run(pT->pTS1);
	pT->pTS2->Run(pT->pTS2);
}
_GLOBAL INT nTSCH;
void CPunit_Processing(This)
{
	DECLARE_MULTI_OPEN(CPunit,CDevice)
}
void CPunit_PostProc(This)
{
	DECLARE_MULTI_OPEN(CPunit,CDevice)
}
/*
typedef struct _tagPUData
{
BYTE bySt0;
BYTE bySt1;
BYTE bySt2;
WORD dwTimeConst;
WORD dwOpenTime;
}SPUDATA;
/*
*/
BOOL CPunit_EventHandler(This,SMESSAGE *pMsg)
{
    DECLARE_MULTI_OPEN(CPunit,CDevice)
	SKPEVENT pEV;
    #ifdef DEB_CPunit
	//Info("\n(%b)CTLSG::>INPT::%M",&pB->m_nCD.wDeviceID,pMsg);
    #endif
	switch(pMsg->m_sbyFor)
	{
	  case DIR_MSTODV:
		   switch(pMsg->m_sbyType)
		   {
		    case PL_DATA_IND:
				 switch(pB->m_nCD.byParam0)
				 {
				   case CTR_TU:
					   switch (pB->m_nCD.byParam1)
					   {
					      case 0:
					         if (pB->m_nCD.wParam0==1) pT->StartPU(pT);else
							 if (pB->m_nCD.wParam0==0) pT->StopPU(pT);
						  break;
						  case 1:
							  if (pB->m_nCD.wParam0==0)
							  {
								pT->pP->sDT.wSt0 &= ~(0x01);
                                pT->pTU0->InvPin(pT->pTU0);
							  }else
							  if (pB->m_nCD.wParam0==1) pT->pP->sDT.wSt0 |=  (0x01);
						  break;
						  default:
						  break;
					   }

                        //#ifdef DEB_CFreq
	                    //Info("\n(%b)CTLSG::>CTR_TR::%d",&pB->m_nCD.wDeviceID,&pB->m_nCD.fParam0);
                        //#endif
				   break;
				   default:
				   break;
				 }
		    break;
			case EV_CHNG_PIN_REQ:
 				 memcpy(&pEV,&pMsg->m_sbyInfo[0],sizeof(SKPEVENT));
				 switch (pEV.byType)
				 {
				    case REG_SOFTU_ADDR:
						if ((pEV.byCause==EV_0T1_ST)&&(pEV.byAddr==0))
							pT->pP->sDT.wSt0 |=  (0x02);else
						if ((pEV.byCause==EV_1T0_ST)&&(pEV.byAddr==0))
							pT->pP->sDT.wSt0 &= ~(0x02);else
					break;
					case REG_SOFTS_ADDR:
						//Активность левого выхода
						if ((pEV.byCause==EV_0T1_CH)&&(pEV.byAddr==0))
							pT->pP->sDT.wSt0 |=  (0x04);else
						if ((pEV.byCause==EV_1T0_CH)&&(pEV.byAddr==0))
							pT->pP->sDT.wSt0 &= ~(0x04);else
						//Активность среднего выхода
						if ((pEV.byCause==EV_0T1_CH)&&(pEV.byAddr==1))
							pT->pP->sDT.wSt0 |=  (0x08);else
						if ((pEV.byCause==EV_1T0_CH)&&(pEV.byAddr==1))
							pT->pP->sDT.wSt0 &= ~(0x08);else
						//Активность левого выхода
						if ((pEV.byCause==EV_0T1_CH)&&(pEV.byAddr==2))
							pT->pP->sDT.wSt0 |=  (0x10);else
						if ((pEV.byCause==EV_1T0_CH)&&(pEV.byAddr==2))
							pT->pP->sDT.wSt0 &= ~(0x10);else
					break;
				 }
			break;
			default:
            break;
		   }
      break;
	  case DIR_101MD:
	  break;
	  default:
	  break;
	}
	return TRUE;
}
void CPunit_StartPU(This)
{
    DECLARE_MULTI_OPEN(CPunit,CDevice)
	if(pT->pP->sDT.wSt0 & 0x01)
	{
     pT->pTU0->SetPin(pT->pTU0);
     #ifdef DEB_CPunit
	 Info("\n(%b)CPUNT::>OPEN PU",&pB->m_nCD.wDeviceID);
     #endif
	}
}
void CPunit_StopPU(This)
{
    DECLARE_MULTI_OPEN(CPunit,CDevice)
	if(pT->pP->sDT.wSt0 & 0x01)
	{
     pT->pTU0->InvPin(pT->pTU0);
     #ifdef DEB_CPunit
	 Info("\n(%b)CPUNT::>CLOSE PU",&pB->m_nCD.wDeviceID);
     #endif
	}
}
void CPunit_ClosePU(This)
{
    DECLARE_MULTI_OPEN(CPunit,CDevice)
    //pT->pP->sDT.wSt0 &= ~(0x01);
    pT->pTU0->InvPin(pT->pTU0);
    #ifdef DEB_CPunit
	Info("\n(%b)CPUNT::>STOP PU",&pB->m_nCD.wDeviceID);
    #endif
}
/*
typedef struct _tagPUData
{
BYTE bySt0;
BYTE bySt1;
BYTE bySt2;
UINT dwTimeConst;
UINT dwOpenTime;
}SPUDATA;
*/
PVOID CPunit_GetData(This,BYTE *pData,WORD *nLen)
{
    DECLARE_MULTI_OPEN(CPunit,CDevice)
	pB->GetWordParam(pB,(BYTE*)&pT->pP->sDT.wSt0,&pData[0]);
	pB->GetWordParam(pB,(BYTE*)&pT->pP->sDT.dwTimeConst,&pData[2]);
	pB->GetWordParam(pB,(BYTE*)&pT->pP->sDT.dwOpenTime,&pData[4]);
	*nLen += pB->m_nSize;if (*nLen>350) *nLen=0;
	return pData;
}
void CPunit_CPunit(This)
{
    DECLARE_MULTI_OPEN(CPunit,CDevice)
	DECLARE_REGISTRATION(CPunit,StartPU)
	DECLARE_REGISTRATION(CPunit,StopPU)
	DECLARE_REGISTRATION(CPunit,ClosePU)
	DECLARE_VIRTUAL_FUNC(CPunit,EventHandler)
	DECLARE_VIRTUAL_FUNC(CPunit,InitTCHN)
	DECLARE_VIRTUAL_FUNC(CPunit,PreProc)
	DECLARE_VIRTUAL_FUNC(CPunit,Processing)
	DECLARE_VIRTUAL_FUNC(CPunit,PostProc)
	DECLARE_VIRTUAL_FUNC(CPunit,GetData)
}
void CPunit_DCPunit(This)
{
	DECLARE_MULTI_OPEN(CPunit,CDevice)
}
DECLARE_MULTI_CREATE(CPunit,CDevice)
```

#### bnrstgate.h
```c
/********************************************************************
 * COPYRIGHT -- Kontora
 ********************************************************************
 * Program: bnrmain
 * File: bnraninput.h
 * Author: Abramenya
 * Created: January 19, 2009
 *******************************************************************/

#ifndef __STGATE_H__
#define __STGATE_H__
#include "typedefs.h"
#include "bnrdevice.h"
#include "bnrpin.h"
#include "bnrdevtu.h"
/*
//Управляемые краны
typedef struct _tagTKParam
{
BYTE byID;
BYTE byAmParam;
BYTE byType;
BYTE bySlot;
BYTE byPin;
BYTE bySlot1;
BYTE byPin1;
BYTE byStOP;
BYTE byStCL;
UINT wMaxOpenTime;
UINT wOpenState;
}STKPARAM;
*/
Class CStGate
{
	 void (*CCStGate)(This);
	 void (*DCStGate)(This);
Public
	 Virtual BOOL (*EventHandler)(This,SMESSAGE *pMsg);
	 Virtual void (*InitTCHN)(This,PVOID psTable);
     Virtual void (*PreProc)(This);
	 Virtual void (*Processing)(This);
     Virtual void (*PostProc)(This);
	 Virtual PVOID (*GetData)(This,BYTE *pData,WORD *nLen);
Public
     void (*Open)(This,REAL fOpenPrc);
	 WORD (*PrcToPulce)(This,REAL fOpenPrc);
	 REAL (*PulceToPrc)(This,DWORD dwPulce);
	 DWORD (*SecToPulce)(This,WORD wOpenTime);
	 BOOL (*GetOpenDir)(This,DWORD dwPulce);
	 WORD (*GetOpenPulce)(This,BOOL blDir,DWORD dwOpenPulce);
	 void (*OpenGate)(This,BOOL blDir,DWORD dwOpenPulce);
Public
     STKPARAM *pP;
     CDevTU *pTU0;
     CDevTU *pTU1;
	 DWORD m_dwOpenState;
	 DWORD m_dwOldJob;
	 DWORD m_dwOpenGate;
	 DWORD m_dwCloseGate;
	 DWORD m_dwPulce;
	 DECLARE_IMPLEMENT_BASE(CDevice)
}
DECLARE_DEFINITION(CStGate)
#endif
```

#### bnrstgate.c
```c
/********************************************************************
 * COPYRIGHT -- Kontora
 ********************************************************************
 * Program: bnrmain
 * File: bnrlsens.c
 * Author: Abramenya
 * Created: January 19, 2009
 *******************************************************************/

#include "bnrstgate.h"
#include "bnrmain.h"
#ifdef _DEFAULT_INCLUDES
 #include <AsDefault.h>
#endif
_GLOBAL BYTE nFSignal;
/*
//Управляемые краны
typedef struct _tagTKParam
{
BYTE byID;
BYTE byAmParam;
BYTE byType;
BYTE bySlot;
BYTE byPin;
BYTE bySlot1;
BYTE byPin1;
BYTE byStOP;
BYTE byStCL;
UINT wMaxOpenTime;
UINT wOpenState;
}STKPARAM;
*/
void CStGate_InitTCHN(This,PVOID psTable)
{
    DECLARE_MULTI_OPEN(CStGate,CDevice)
	BOOL  *m_pbVL;
	CSlot *pSL;
	CPin  *m_pPN;
	CComputer *pCM = pB->m_pComputer;
	pT->pP         = (STKPARAM*)psTable;
	pB->m_nSize    = 3+sizeof(WORD)+2*sizeof(REAL);

    pT->m_dwOpenState = 0;
	pT->m_dwOldJob    = 0;

	//Выход Открытия
	pSL    = pCM->GetSlot(pCM,pT->pP->bySlot);
	m_pPN  = pSL->GetPin(pSL->pChld,pT->pP->byPin);
    m_pbVL = (BOOL*)m_pPN->GetAddrPin(m_pPN->pChld);
	New(sizeof(CDevTU),pT->pTU0);
	InitObject(CDevTU,pT->pTU0);
    pT->pTU0->Init(pT->pTU0,m_pbVL,pT->pP->byID,0,EN_OPEN,EN_DIRECT,100);
	pT->pTU0->SetTU(pT->pTU0,DEV_MSMDL_BOX_ID,DIR_MSTOMS,EV_CHNG_PIN_REQ);

	//Выход Закрытия
	pSL     = pCM->GetSlot(pCM,pT->pP->bySlot1);
	m_pPN  = pSL->GetPin(pSL->pChld,pT->pP->byPin1);
    m_pbVL = (BOOL*)m_pPN->GetAddrPin(m_pPN->pChld);
	New(sizeof(CDevTU),pT->pTU1);
	InitObject(CDevTU,pT->pTU1);
    pT->pTU1->Init(pT->pTU1,m_pbVL,pT->pP->byID,1,EN_OPEN,EN_DIRECT,100);
	pT->pTU1->SetTU(pT->pTU1,DEV_MSMDL_BOX_ID,DIR_MSTOMS,EV_CHNG_PIN_REQ);

    #ifdef DEB_CStGate
	//Info("\n(%b)CTLSG::>Create TeleSignal.",&pB->m_byID);
    #endif
}
void CStGate_PreProc(This)
{
    DECLARE_MULTI_OPEN(CStGate,CDevice)
	pT->m_dwOpenGate  = pT->pTU0->Run(pT->pTU0);
	pT->m_dwCloseGate = pT->pTU1->Run(pT->pTU1);
}
void CStGate_Processing(This)
{
	DECLARE_MULTI_OPEN(CStGate,CDevice)
}
void CStGate_PostProc(This)
{
	DECLARE_MULTI_OPEN(CStGate,CDevice)
}
/*
typedef struct _tagTKData
{
BYTE byStOP;
BYTE byStCL;
WORD wMaxOpenTime;
REAL fJobOpen;
REAL fOpenState;
}STKDATA;
*/
BOOL CStGate_EventHandler(This,SMESSAGE *pMsg)
{
    DECLARE_MULTI_OPEN(CStGate,CDevice)
	SKPEVENT pEV;
    #ifdef DEB_CStGate
	//Info("\n(%b)CTLSG::>INPT::%M",&pB->m_nCD.wDeviceID,pMsg);
    #endif
	switch(pMsg->m_sbyFor)
	{
	  case DIR_MSTODV:
		   switch(pMsg->m_sbyType)
		   {
		    case PL_DATA_IND:
                 switch(pB->m_nCD.byParam0)
				 {
				   case CTR_TR:
					    switch (pB->m_nCD.byParam1)
					    {
						  case 0:
							  if (pT->m_dwOpenState==0) pT->pP->sDT.wMaxOpenTime = (WORD)(pB->m_nCD.fParam0);
						  break;
						  case 1:
							  if ((pB->m_nCD.fParam0>=0.0)&&(pB->m_nCD.fParam0<=100.0))
							  {
							   pT->pP->sDT.byStMD   = 1;
							   pT->pP->sDT.fJobOpen = pB->m_nCD.fParam0;
							   pT->Open(pT,pT->pP->sDT.fJobOpen);
							  }
						  break;
						  default:
						  break;
					    }
				   break;
				   case CTR_TU:
					   if (pB->m_nCD.wParam0==1)
					   {
						 //pT->pTU0->SetPulce(pT->pTU0);
					   } else
					   if (pB->m_nCD.wParam0==0)
					   {
						 //pT->pTU1->SetPulce(pT->pTU1);
					   }
				   break;
				   case CTR_STOP:
					    pT->m_dwOpenState = pT->m_dwOldJob+pT->m_dwOpenGate-pT->m_dwCloseGate;
						pT->pTU0->Stop(pT->pTU0);
						pT->pTU1->Stop(pT->pTU1);
                        #ifdef DEB_CStGate
	                    Info("\n(%b)CSTGT::>STOP GATE",&pB->m_nCD.wDeviceID);
                        #endif
				   break;
				   case CTR_OPEN:
					    pT->Open(pT,pB->m_nCD.fParam0);
                        #ifdef DEB_CStGate
	                    Info("\n(%b)CSTGT::>OPEN GATE",&pB->m_nCD.wDeviceID);
                        #endif
				   break;
				   case CTR_CLOSE:
						pT->Open(pT,pB->m_nCD.fParam0);
                        #ifdef DEB_CStGate
	                    Info("\n(%b)CSTGT::>CLOSE GATE",&pB->m_nCD.wDeviceID);
                        #endif
				   break;
				   default:
				   break;
				 }
		    break;
			case EV_CHNG_PIN_REQ:
 				 memcpy(&pEV,&pMsg->m_sbyInfo[0],sizeof(SKPEVENT));
				 switch (pEV.byType)
				 {
				    case REG_SOFTU_ADDR:
						//Состояние открытия
						if ((pEV.byCause==EV_0T1_ST)&&(pEV.byAddr==0))
						{
						 pT->pP->sDT.byStOP = 1;
						 #ifdef DEB_CStGate
						 Info("\n(%b)CSTGT::>START OPEN(%d)",&pB->m_nCD.wDeviceID,&pT->m_dwPulce);
                         #endif
						} else
						if ((pEV.byCause==EV_1T0_ST)&&(pEV.byAddr==0))
						{
						 pT->pP->sDT.byStOP     = 0;
						 pT->pP->sDT.fOpenState = pT->PulceToPrc(pT,pT->m_dwOpenState);
						 pT->m_dwOldJob         = pT->m_dwOpenState;
						 if (pT->pP->sDT.byStMD==1) pT->pP->sDT.byStMD = 0;
						 #ifdef DEB_CStGate
						 Info("\n(%b)CSTGT::>STOP  OPEN(%d)",&pB->m_nCD.wDeviceID,&pT->m_dwPulce);
                         #endif
						} else
                        //Состояние закрытия
						if ((pEV.byCause==EV_0T1_ST)&&(pEV.byAddr==1))
						{
						 pT->pP->sDT.byStCL = 1;
						 #ifdef DEB_CStGate
						 Info("\n(%b)CSTGT::>START CLOSE(%d)",&pB->m_nCD.wDeviceID,&pT->m_dwPulce);
                         #endif
						} else
						if ((pEV.byCause==EV_1T0_ST)&&(pEV.byAddr==1))
						{
						 pT->pP->sDT.byStCL     = 0;
						 pT->pP->sDT.fOpenState = pT->PulceToPrc(pT,pT->m_dwOpenState);
						 pT->m_dwOldJob         = pT->m_dwOpenState;
						 if (pT->pP->sDT.byStMD==1) pT->pP->sDT.byStMD = 0;
						 #ifdef DEB_CStGate
						 Info("\n(%b)CSTGT::>STOP  CLOSE(%d)",&pB->m_nCD.wDeviceID,&pT->m_dwPulce);
                         #endif
						}
					break;
					case REG_SOFTS_ADDR:
						//Активность с релейного выхода
						//if ((pEV.byCause==EV_0T1_CH)&&(pEV.byAddr==0))
						//	pT->pP->sDT.byAlST0 = 1;
						//if ((pEV.byCause==EV_1T0_CH)&&(pEV.byAddr==0))
						//	pT->pP->sDT.byAlST0 = 0;
						//Авария
						//if ((pEV.byCause==EV_0T1_CH)&&(pEV.byAddr==1))
						//	pT->pP->sDT.byAlST1 = 1;
						//if ((pEV.byCause==EV_1T0_CH)&&(pEV.byAddr==1))
						//	pT->pP->sDT.byAlST1 = 0;
					break;
				 }
			break;
			default:
            break;
		   }
      break;
	  case DIR_101MD:
	  break;
	  default:
	  break;
	}
	return TRUE;
}
void CStGate_Open(This,REAL fOpenPrc)
{
    DECLARE_MULTI_OPEN(CStGate,CDevice)
	DWORD dwPulce = pT->PrcToPulce(pT,fOpenPrc);
	BOOL  blDir   = pT->GetOpenDir(pT,dwPulce);
	DWORD nOPulce = pT->GetOpenPulce(pT,blDir,dwPulce);
	pT->m_dwPulce = nOPulce; //для отладки
	if (pT->m_dwOpenState==dwPulce) return;
	pT->m_dwOpenState = dwPulce;
	pT->OpenGate(pT,blDir,nOPulce);
}
DWORD CStGate_PrcToPulce(This,REAL fOpenPrc)
{
    DECLARE_MULTI_OPEN(CStGate,CDevice)
	REAL fTime     = (REAL)(1000*pT->pP->sDT.wMaxOpenTime);
	REAL fOpen     = (REAL)(fOpenPrc/100.0);
	REAL fSysQuant = (REAL)SYSTEM_QTIME;
    DWORD dwPulce  = (DWORD)(fTime*fOpen/fSysQuant);
    return dwPulce;
}
REAL CStGate_PulceToPrc(This,DWORD dwPulce)
{
    DECLARE_MULTI_OPEN(CStGate,CDevice)
	REAL fTime     = (REAL)(1000*pT->pP->sDT.wMaxOpenTime);
	REAL fSysQuant = (REAL)SYSTEM_QTIME;
	REAL fPulce    = (REAL)dwPulce;
	REAL fOpen     = (REAL)(100.0*fPulce/(fTime/fSysQuant));
    return fOpen;
}
DWORD CStGate_SecToPulce(This,WORD wOpenTime)
{
    DECLARE_MULTI_OPEN(CStGate,CDevice)
	REAL fTime     = (REAL)(1000*wOpenTime);
	REAL fSysQuant = (REAL)SYSTEM_QTIME;
    DWORD dwPulce  = (DWORD)(fTime/fSysQuant);
    return dwPulce;
}
BOOL CStGate_GetOpenDir(This,DWORD dwPulce)
{
    DECLARE_MULTI_OPEN(CStGate,CDevice)
	BOOL res = FALSE;
    if (dwPulce>=pT->m_dwOpenState) res = TRUE; else
    if (dwPulce<pT->m_dwOpenState)  res = FALSE;
	return res;
}
DWORD CStGate_GetOpenPulce(This,BOOL blDir,DWORD dwOpenPulce)
{
    DECLARE_MULTI_OPEN(CStGate,CDevice)
	DWORD dwPulce=0;
	if (blDir==TRUE)
     dwPulce = (dwOpenPulce-pT->m_dwOpenState); else
	if (blDir==FALSE)
	 dwPulce = (pT->m_dwOpenState-dwOpenPulce);
    return dwPulce;
}
void CStGate_OpenGate(This,BOOL blDir,DWORD dwOpenPulce)
{
    DECLARE_MULTI_OPEN(CStGate,CDevice)
	if (blDir==TRUE)
  	 pT->pTU0->SetPulceEx(pT->pTU0,dwOpenPulce);
	if (blDir==FALSE)
	 pT->pTU1->SetPulceEx(pT->pTU1,dwOpenPulce);
}
/*
typedef struct _tagTKData
{
	BYTE byStOP;
	BYTE byStCL;
    WORD wMaxOpenTime;
    REAL fJobOpen;
    REAL fOpenState;
}STKDATA;
*/
PVOID CStGate_GetData(This,BYTE *pData,WORD *nLen)
{
    DECLARE_MULTI_OPEN(CStGate,CDevice)
	pData[0] = pT->pP->sDT.byStOP;
	pData[1] = pT->pP->sDT.byStCL;
	pData[2] = pT->pP->sDT.byStMD;
	pB->GetWordParam(pB,(BYTE*)&pT->pP->sDT.wMaxOpenTime,&pData[3]);
	pB->GetRealParam(pB,(BYTE*)&pT->pP->sDT.fJobOpen,&pData[5]);
	pB->GetRealParam(pB,(BYTE*)&pT->pP->sDT.fOpenState,&pData[9]);
	*nLen += pB->m_nSize;if (*nLen>350) *nLen=0;
	pT->pP->sDT.fOpenState = pT->PulceToPrc(pT,pT->m_dwOldJob+pT->m_dwOpenGate-pT->m_dwCloseGate);
	return pData;
}
void CStGate_CStGate(This)
{
    DECLARE_MULTI_OPEN(CStGate,CDevice)
	DECLARE_REGISTRATION(CStGate,Open)
	DECLARE_REGISTRATION(CStGate,PrcToPulce)
	DECLARE_REGISTRATION(CStGate,PulceToPrc)
	DECLARE_REGISTRATION(CStGate,SecToPulce)
	DECLARE_REGISTRATION(CStGate,GetOpenDir)
	DECLARE_REGISTRATION(CStGate,GetOpenPulce)
	DECLARE_REGISTRATION(CStGate,OpenGate)
	DECLARE_VIRTUAL_FUNC(CStGate,EventHandler)
	DECLARE_VIRTUAL_FUNC(CStGate,InitTCHN)
	DECLARE_VIRTUAL_FUNC(CStGate,PreProc)
	DECLARE_VIRTUAL_FUNC(CStGate,Processing)
	DECLARE_VIRTUAL_FUNC(CStGate,PostProc)
	DECLARE_VIRTUAL_FUNC(CStGate,GetData)
}
void CStGate_DCStGate(This)
{
	DECLARE_MULTI_OPEN(CStGate,CDevice)
}
DECLARE_MULTI_CREATE(CStGate,CDevice)
```

#### bnrtcpserver.h
```c
/********************************************************************
 * COPYRIGHT -- Kontora
 ********************************************************************
 * Program: bnrmain
 * File: bnraninput.h
 * Author: Abramenya
 * Created: January 19, 2009
 *******************************************************************/

#ifndef __TCPSERVER_H__
#define __TCPSERVER_H__
#include "typedefs.h"
#include "bnrmessage.h"
#include "bnrdebug.h"
#include "bnrpob.h"
#include "bnrcyclicsystem.h"
#ifdef WIN32
#include "AsTCP1.h"
#include "winsock.h"
#else
//#include <Ethernet.h>
#endif
Class CTcpServer
{
	 void (*CCTcpServer)(This);
	 void (*DCTcpServer)(This);
Public
     //Connection Disconnection Procedure
     void (*Init)(This,SARMINTERFACE *pArm);
     BOOL (*SendMessage)(This,SMESSAGE *pMsg);
	 BOOL (*GetMessage)(This,SMESSAGE *pMsg);
Private
	 BOOL (*Open)(This);
	 BOOL (*Listen)(This);
	 BOOL (*Close)(This,UDINT uModule);
	 BOOL (*CloseSend)(This);
	 BOOL (*CloseRecc)(This);
	 BOOL (*CheckSend)(This);
	 BOOL (*CloseOpen)(This);
	 void (*PostSend)(This);
	 BOOL (*PostGet)(This);
	 void (*WordXCHG)(This,SMESSAGE *pMsg);
	 BOOL (*CheckCRC)(This,BOOL,SMESSAGE *pMsg);
     void (*AddCRC)(This,BOOL,SMESSAGE *pMsg);
	 BOOL (*Connect)(This);
	 BOOL (*Disconnect)(This);
	 void (*SendSMessage)(This,BYTE byBox,BYTE byFor,BYTE byType);
	 DWORD (*ClcCRC)(This,BOOL,SMESSAGE *pMsg);
	 void (*ReceiveThread)(This);
	 void (*SendThread)(This);
	 Virtual BOOL (*EventHandler)(This,SMESSAGE *pMsg);
     Virtual void (*CyclicProc)(This);
Private
     SARMINTERFACE *m_pArm;
	 TcpServer_typ m_npServer;
     TcpOpen_typ m_npListen;
     TcpSend_typ m_npSend;
	 TcpRecv_typ m_npRecc;
     TcpClose_typ m_npClose;
     BOOL m_blSState;
	 BOOL m_blRState;
     DWORD m_dwAPortNumber;
	 DWORD m_dwBPortNumber;
     char m_stTcpAddr[50];
	 BYTE m_bSrvState;
	 BYTE m_bCliState;
	 BYTE m_byConnReq;
	 SMESSAGE m_sMsg;
	 SMESSAGE m_sMsg0;
	 CMTimer m_nConnTMR;
	 DECLARE_IMPLEMENT_BASE(CCyclicSystem)
}
DECLARE_DEFINITION(CTcpServer)
#endif
```
